LIN {X 0,Y 410.972,Z 398.401,A -85,B 0,C 180,E1 -10552.131,E2 -10552.131} C_VEL
LIN {X 0,Y 410.999,Z 397.235,A -85,B 0,C 180,E1 -10552.341,E2 -10552.341} C_VEL
LIN {X 0,Y 411.344,Z 382.792,A -85,B 0,C 180,E1 -10556.102,E2 -10556.102} C_VEL
LIN {X 0,Y 411.817,Z 369.639,A -85,B 0,C 180,E1 -10559.664,E2 -10559.664} C_VEL
LIN {X 0,Y 412.354,Z 356.779,A -85,B 0,C 180,E1 -10563.37,E2 -10563.37} C_VEL
LIN {X 0,Y 413.561,Z 344.278,A -85,B 0,C 180,E1 -10567.276,E2 -10567.276} C_VEL
LIN {X 0,Y 414.274,Z 339.521,A -85,B 0,C 180,E1 -10568.881,E2 -10568.881} C_VEL
LIN {X 0,Y 414.062,Z 336.041,A -85,B 0,C 180,E1 -10570.2,E2 -10570.2} C_VEL
LIN {X 0,Y 412.867,Z 329.754,A -85,B 0,C 180,E1 -10572.949,E2 -10572.949} C_VEL
LIN {X 0,Y 411.688,Z 324.313,A -85,B 0,C 180,E1 -10575.807,E2 -10575.807} C_VEL
LIN {X 0,Y 411.209,Z 321.929,A -85,B 0,C 180,E1 -10577.301,E2 -10577.301} C_VEL
LIN {X 0,Y 411.234,Z 321.886,A -85,B 0,C 180,E1 -10580.778,E2 -10580.778} C_VEL
LIN {X 0,Y 411.203,Z 321.888,A -85,B 0,C 180,E1 -10584.472,E2 -10584.472} C_VEL
LIN {X 0,Y 411.21,Z 321.889,A -85,B 0,C 180,E1 -10586.874,E2 -10586.874} C_VEL
LIN {X 0,Y 411.236,Z 321.885,A -85,B 0,C 180,E1 -10590.645,E2 -10590.645} C_VEL
LIN {X 0,Y 411.241,Z 321.886,A -85,B 0,C 180,E1 -10593.62,E2 -10593.62} C_VEL
LIN {X 0,Y 411.207,Z 321.891,A -85,B 0,C 180,E1 -10596.853,E2 -10596.853} C_VEL
LIN {X 0,Y 411.235,Z 322.056,A -85,B 0,C 180,E1 -10597.53,E2 -10597.53} C_VEL
LIN {X 0,Y 411.571,Z 323.361,A -85,B 0,C 180,E1 -10597.754,E2 -10597.754} C_VEL
LIN {X 0,Y 416.935,Z 335.703,A -85,B 0,C 180,E1 -10598.946,E2 -10598.946} C_VEL
LIN {X 0,Y 419.583,Z 343.599,A -85,B 0,C 180,E1 -10599.719,E2 -10599.719} C_VEL
LIN {X 0,Y 418.83,Z 355.331,A -85,B 0,C 180,E1 -10600.646,E2 -10600.646} C_VEL
LIN {X 0,Y 417.749,Z 367.989,A -85,B 0,C 180,E1 -10601.867,E2 -10601.867} C_VEL
LIN {X 0,Y 416.783,Z 378.362,A -85,B 0,C 180,E1 -10603.09,E2 -10603.09} C_VEL
LIN {X 0,Y 415.804,Z 388.025,A -85,B 0,C 180,E1 -10604.457,E2 -10604.457} C_VEL
LIN {X 0,Y 414.968,Z 394.51,A -85,B 0,C 180,E1 -10605.534,E2 -10605.534} C_VEL
LIN {X 0,Y 414.04,Z 403.147,A -85,B 0,C 180,E1 -10607.252,E2 -10607.252} C_VEL
LIN {X 0,Y 413.307,Z 409.172,A -85,B 0,C 180,E1 -10608.723,E2 -10608.723} C_VEL
LIN {X 0,Y 412.749,Z 414.131,A -85,B 0,C 180,E1 -10610.197,E2 -10610.197} C_VEL
LIN {X 0,Y 412.146,Z 419.249,A -85,B 0,C 180,E1 -10612.16,E2 -10612.16} C_VEL
LIN {X 0,Y 411.574,Z 422.875,A -85,B 0,C 180,E1 -10614.12,E2 -10614.12} C_VEL
LIN {X 0,Y 411.29,Z 425.054,A -85,B 0,C 180,E1 -10616.081,E2 -10616.081} C_VEL
LIN {X 0,Y 411.179,Z 425.847,A -85,B 0,C 180,E1 -10618.041,E2 -10618.041} C_VEL
LIN {X 0,Y 411.073,Z 425.319,A -85,B 0,C 180,E1 -10620,E2 -10620} C_VEL
LIN {X 0,Y 411.066,Z 423.45,A -85,B 0,C 180,E1 -10621.96,E2 -10621.96} C_VEL
LIN {X 0,Y 411.103,Z 420.216,A -85,B 0,C 180,E1 -10623.921,E2 -10623.921} C_VEL
LIN {X 0,Y 411.471,Z 415.498,A -85,B 0,C 180,E1 -10625.882,E2 -10625.882} C_VEL
LIN {X 0,Y 411.831,Z 410.884,A -85,B 0,C 180,E1 -10627.354,E2 -10627.354} C_VEL
LIN {X 0,Y 412.243,Z 404.257,A -85,B 0,C 180,E1 -10629.073,E2 -10629.073} C_VEL
LIN {X 0,Y 412.88,Z 396.057,A -85,B 0,C 180,E1 -10630.792,E2 -10630.792} C_VEL
LIN {X 0,Y 413.504,Z 387.517,A -85,B 0,C 180,E1 -10632.266,E2 -10632.266} C_VEL
LIN {X 0,Y 414.234,Z 377.269,A -85,B 0,C 180,E1 -10633.741,E2 -10633.741} C_VEL
LIN {X 0,Y 415.128,Z 365.737,A -85,B 0,C 180,E1 -10635.099,E2 -10635.099} C_VEL
LIN {X 0,Y 415.874,Z 353.184,A -85,B 0,C 180,E1 -10636.317,E2 -10636.317} C_VEL
LIN {X 0,Y 416.618,Z 341.348,A -85,B 0,C 180,E1 -10637.253,E2 -10637.253} C_VEL
LIN {X 0,Y 416.273,Z 338.757,A -85,B 0,C 180,E1 -10637.46,E2 -10637.46} C_VEL
LIN {X 0,Y 412.31,Z 325.603,A -85,B 0,C 180,E1 -10638.462,E2 -10638.462} C_VEL
LIN {X 0,Y 411.361,Z 322.465,A -85,B 0,C 180,E1 -10638.716,E2 -10638.716} C_VEL
LIN {X 0,Y 411.252,Z 321.899,A -85,B 0,C 180,E1 -10638.948,E2 -10638.948} C_VEL
LIN {X 0,Y 411.209,Z 321.891,A -85,B 0,C 180,E1 -10642.643,E2 -10642.643} C_VEL
LIN {X 0,Y 411.241,Z 321.881,A -85,B 0,C 180,E1 -10645.293,E2 -10645.293} C_VEL
LIN {X 0,Y 411.264,Z 321.877,A -85,B 0,C 180,E1 -10647.478,E2 -10647.478} C_VEL
LIN {X 0,Y 411.195,Z 321.89,A -85,B 0,C 180,E1 -10650.848,E2 -10650.848} C_VEL
LIN {X 0,Y 411.211,Z 321.888,A -85,B 0,C 180,E1 -10654.333,E2 -10654.333} C_VEL
LIN {X 0,Y 411.197,Z 321.887,A -85,B 0,C 180,E1 -10657.974,E2 -10657.974} C_VEL
LIN {X 0,Y 411.168,Z 321.889,A -85,B 0,C 180,E1 -10661.228,E2 -10661.228} C_VEL
LIN {X 0,Y 411.182,Z 321.894,A -85,B 0,C 180,E1 -10664.49,E2 -10664.49} C_VEL
LIN {X 0,Y 411.203,Z 321.89,A -85,B 0,C 180,E1 -10668.197,E2 -10668.197} C_VEL
LIN {X 0,Y 411.23,Z 321.884,A -85,B 0,C 180,E1 -10670.776,E2 -10670.776} C_VEL
LIN {X 0,Y 411.204,Z 321.889,A -85,B 0,C 180,E1 -10674.471,E2 -10674.471} C_VEL
LIN {X 0,Y 411.213,Z 321.884,A -85,B 0,C 180,E1 -10676.873,E2 -10676.873} C_VEL
LIN {X 0,Y 411.239,Z 321.882,A -85,B 0,C 180,E1 -10680.644,E2 -10680.644} C_VEL
LIN {X 0,Y 411.243,Z 321.881,A -85,B 0,C 180,E1 -10683.619,E2 -10683.619} C_VEL
LIN {X 0,Y 411.202,Z 321.885,A -85,B 0,C 180,E1 -10686.852,E2 -10686.852} C_VEL
LIN {X 0,Y 411.222,Z 321.89,A -85,B 0,C 180,E1 -10690.049,E2 -10690.049} C_VEL
LIN {X 0,Y 411.269,Z 321.877,A -85,B 0,C 180,E1 -10693.131,E2 -10693.131} C_VEL
LIN {X 0,Y 411.311,Z 321.871,A -85,B 0,C 180,E1 -10696.895,E2 -10696.895} C_VEL
LIN {X 0,Y 411.298,Z 321.877,A -85,B 0,C 180,E1 -10700.161,E2 -10700.161} C_VEL
LIN {X 0,Y 411.488,Z 321.853,A -85,B 0,C 180,E1 -10702.146,E2 -10702.146} C_VEL
LIN {X 0,Y 411.478,Z 321.854,A -85,B 0,C 180,E1 -10704.117,E2 -10704.117} C_VEL
LIN {X 0,Y 411.516,Z 321.85,A -85,B 0,C 180,E1 -10708.042,E2 -10708.042} C_VEL
LIN {X 0,Y 411.645,Z 321.834,A -85,B 0,C 180,E1 -10709.999,E2 -10709.999} C_VEL
LIN {X 0,Y 411.463,Z 321.853,A -85,B 0,C 180,E1 -10712.936,E2 -10712.936} C_VEL
LIN {X 0,Y 411.465,Z 321.852,A -85,B 0,C 180,E1 -10716.866,E2 -10716.866} C_VEL
LIN {X 0,Y 411.297,Z 321.877,A -85,B 0,C 180,E1 -10719.838,E2 -10719.838} C_VEL
LIN {X 0,Y 411.291,Z 321.874,A -85,B 0,C 180,E1 -10722.601,E2 -10722.601} C_VEL
LIN {X 0,Y 410.65,Z 321.959,A -85,B 0,C 180,E1 -10723.419,E2 -10723.419} C_VEL
LIN {X 0,Y 407.769,Z 322.313,A -85,B 0,C 180,E1 -10724.745,E2 -10724.745} C_VEL
LIN {X 0,Y 405.323,Z 322.621,A -85,B 0,C 180,E1 -10725.817,E2 -10725.817} C_VEL
LIN {X 0,Y 404.289,Z 322.747,A -85,B 0,C 180,E1 -10726.647,E2 -10726.647} C_VEL
LIN {X 0,Y 404.215,Z 322.757,A -85,B 0,C 180,E1 -10726.928,E2 -10726.928} C_VEL
LIN {X 0,Y 404.166,Z 322.761,A -85,B 0,C 180,E1 -10730.35,E2 -10730.35} C_VEL
LIN {X 0,Y 404.171,Z 322.766,A -85,B 0,C 180,E1 -10733.573,E2 -10733.573} C_VEL
LIN {X 0,Y 404.185,Z 322.762,A -85,B 0,C 180,E1 -10735.765,E2 -10735.765} C_VEL
LIN {X 0,Y 404.195,Z 322.758,A -85,B 0,C 180,E1 -10737.998,E2 -10737.998} C_VEL
LIN {X 0,Y 404.139,Z 322.768,A -85,B 0,C 180,E1 -10741.557,E2 -10741.557} C_VEL
LIN {X 0,Y 404.183,Z 322.764,A -85,B 0,C 180,E1 -10745.015,E2 -10745.015} C_VEL
LIN {X 0,Y 404.154,Z 322.766,A -85,B 0,C 180,E1 -10748.756,E2 -10748.756} C_VEL
LIN {X 0,Y 404.122,Z 322.769,A -85,B 0,C 180,E1 -10751.599,E2 -10751.599} C_VEL
LIN {X 0,Y 404.147,Z 322.765,A -85,B 0,C 180,E1 -10754.522,E2 -10754.522} C_VEL
LIN {X 0,Y 404.136,Z 322.769,A -85,B 0,C 180,E1 -10757.295,E2 -10757.295} C_VEL
LIN {X 0,Y 404.164,Z 322.761,A -85,B 0,C 180,E1 -10759.954,E2 -10759.954} C_VEL
LIN {X 0,Y 404.136,Z 322.77,A -85,B 0,C 180,E1 -10763.123,E2 -10763.123} C_VEL
LIN {X 0,Y 404.14,Z 322.765,A -85,B 0,C 180,E1 -10766.187,E2 -10766.187} C_VEL
LIN {X 0,Y 404.151,Z 322.763,A -85,B 0,C 180,E1 -10769.715,E2 -10769.715} C_VEL
LIN {X 0,Y 404.189,Z 322.762,A -85,B 0,C 180,E1 -10773.122,E2 -10773.122} C_VEL
LIN {X 0,Y 404.171,Z 322.762,A -85,B 0,C 180,E1 -10775.334,E2 -10775.334} C_VEL
LIN {X 0,Y 404.153,Z 322.769,A -85,B 0,C 180,E1 -10778.581,E2 -10778.581} C_VEL
LIN {X 0,Y 404.203,Z 322.757,A -85,B 0,C 180,E1 -10781.761,E2 -10781.761} C_VEL
LIN {X 0,Y 404.2,Z 322.761,A -85,B 0,C 180,E1 -10784.881,E2 -10784.881} C_VEL
LIN {X 0,Y 404.249,Z 322.752,A -85,B 0,C 180,E1 -10787.958,E2 -10787.958} C_VEL
LIN {X 0,Y 404.425,Z 322.732,A -85,B 0,C 180,E1 -10792.099,E2 -10792.099} C_VEL
LIN {X 0,Y 404.416,Z 322.732,A -85,B 0,C 180,E1 -10794.015,E2 -10794.015} C_VEL
LIN {X 0,Y 404.475,Z 322.725,A -85,B 0,C 180,E1 -10798.008,E2 -10798.008} C_VEL
LIN {X 0,Y 404.603,Z 322.71,A -85,B 0,C 180,E1 -10800,E2 -10800} C_VEL
LIN {X 0,Y 404.416,Z 322.731,A -85,B 0,C 180,E1 -10802.988,E2 -10802.988} C_VEL
LIN {X 0,Y 404.403,Z 322.732,A -85,B 0,C 180,E1 -10806.987,E2 -10806.987} C_VEL
LIN {X 0,Y 404.263,Z 322.754,A -85,B 0,C 180,E1 -10810.011,E2 -10810.011} C_VEL
LIN {X 0,Y 404.258,Z 322.75,A -85,B 0,C 180,E1 -10813.211,E2 -10813.211} C_VEL
LIN {X 0,Y 404.21,Z 322.756,A -85,B 0,C 180,E1 -10817.009,E2 -10817.009} C_VEL
LIN {X 0,Y 404.155,Z 322.766,A -85,B 0,C 180,E1 -10820.352,E2 -10820.352} C_VEL
LIN {X 0,Y 404.162,Z 322.764,A -85,B 0,C 180,E1 -10823.575,E2 -10823.575} C_VEL
LIN {X 0,Y 404.176,Z 322.765,A -85,B 0,C 180,E1 -10825.767,E2 -10825.767} C_VEL
LIN {X 0,Y 404.19,Z 322.765,A -85,B 0,C 180,E1 -10828,E2 -10828} C_VEL
LIN {X 0,Y 404.14,Z 322.768,A -85,B 0,C 180,E1 -10831.56,E2 -10831.56} C_VEL
LIN {X 0,Y 404.179,Z 322.76,A -85,B 0,C 180,E1 -10835.017,E2 -10835.017} C_VEL
LIN {X 0,Y 404.157,Z 322.767,A -85,B 0,C 180,E1 -10838.756,E2 -10838.756} C_VEL
LIN {X 0,Y 404.191,Z 322.962,A -85,B 0,C 180,E1 -10842.326,E2 -10842.326} C_VEL
LIN {X 0,Y 406.394,Z 333.763,A -85,B 0,C 180,E1 -10846.234,E2 -10846.234} C_VEL
LIN {X 0,Y 408.182,Z 342.533,A -85,B 0,C 180,E1 -10849.251,E2 -10849.251} C_VEL
LIN {X 0,Y 408.476,Z 347.13,A -85,B 0,C 180,E1 -10850.736,E2 -10850.736} C_VEL
LIN {X 0,Y 407.187,Z 360.221,A -85,B 0,C 180,E1 -10854.725,E2 -10854.725} C_VEL
LIN {X 0,Y 406.079,Z 373.732,A -85,B 0,C 180,E1 -10858.722,E2 -10858.722} C_VEL
LIN {X 0,Y 405.3,Z 385.351,A -85,B 0,C 180,E1 -10862.085,E2 -10862.085} C_VEL
LIN {X 0,Y 404.686,Z 396.904,A -85,B 0,C 180,E1 -10865.369,E2 -10865.369} C_VEL
LIN {X 0,Y 404.088,Z 408.948,A -85,B 0,C 180,E1 -10868.704,E2 -10868.704} C_VEL
LIN {X 0,Y 404.387,Z 411.516,A -85,B 0,C 180,E1 -10868.832,E2 -10868.832} C_VEL
LIN {X 0,Y 406.377,Z 426.794,A -85,B 0,C 180,E1 -10869.406,E2 -10869.406} C_VEL
LIN {X 0,Y 407.897,Z 440.761,A -85,B 0,C 180,E1 -10870.107,E2 -10870.107} C_VEL
LIN {X 0,Y 408.676,Z 451.116,A -85,B 0,C 180,E1 -10870.734,E2 -10870.734} C_VEL
LIN {X 0,Y 407.683,Z 464.047,A -85,B 0,C 180,E1 -10871.639,E2 -10871.639} C_VEL
LIN {X 0,Y 406.699,Z 477.124,A -85,B 0,C 180,E1 -10872.788,E2 -10872.788} C_VEL
LIN {X 0,Y 405.639,Z 488.756,A -85,B 0,C 180,E1 -10874.036,E2 -10874.036} C_VEL
LIN {X 0,Y 404.825,Z 499.405,A -85,B 0,C 180,E1 -10875.421,E2 -10875.421} C_VEL
LIN {X 0,Y 404.157,Z 509.073,A -85,B 0,C 180,E1 -10876.936,E2 -10876.936} C_VEL
LIN {X 0,Y 403.711,Z 518.347,A -85,B 0,C 180,E1 -10878.707,E2 -10878.707} C_VEL
LIN {X 0,Y 403.467,Z 525.787,A -85,B 0,C 180,E1 -10880.476,E2 -10880.476} C_VEL
LIN {X 0,Y 403.415,Z 530.976,A -85,B 0,C 180,E1 -10881.99,E2 -10881.99} C_VEL
LIN {X 0,Y 403.447,Z 534.312,A -85,B 0,C 180,E1 -10883.184,E2 -10883.184} C_VEL
LIN {X 0,Y 403.524,Z 538.294,A -85,B 0,C 180,E1 -10885.005,E2 -10885.005} C_VEL
LIN {X 0,Y 403.583,Z 539.923,A -85,B 0,C 180,E1 -10886.007,E2 -10886.007} C_VEL
LIN {X 0,Y 403.624,Z 542.027,A -85,B 0,C 180,E1 -10888.005,E2 -10888.005} C_VEL
LIN {X 0,Y 403.866,Z 542.674,A -85,B 0,C 180,E1 -10890.001,E2 -10890.001} C_VEL
LIN {X 0,Y 403.853,Z 542.423,A -85,B 0,C 180,E1 -10890.998,E2 -10890.998} C_VEL
LIN {X 0,Y 403.643,Z 540.784,A -85,B 0,C 180,E1 -10892.995,E2 -10892.995} C_VEL
LIN {X 0,Y 403.665,Z 539.422,A -85,B 0,C 180,E1 -10893.994,E2 -10893.994} C_VEL
LIN {X 0,Y 403.584,Z 536.612,A -85,B 0,C 180,E1 -10895.497,E2 -10895.497} C_VEL
LIN {X 0,Y 403.484,Z 532.933,A -85,B 0,C 180,E1 -10897.004,E2 -10897.004} C_VEL
LIN {X 0,Y 403.459,Z 528.291,A -85,B 0,C 180,E1 -10898.516,E2 -10898.516} C_VEL
LIN {X 0,Y 403.529,Z 521.585,A -85,B 0,C 180,E1 -10900.284,E2 -10900.284} C_VEL
LIN {X 0,Y 403.865,Z 513.357,A -85,B 0,C 180,E1 -10902.054,E2 -10902.054} C_VEL
LIN {X 0,Y 404.348,Z 505.162,A -85,B 0,C 180,E1 -10903.52,E2 -10903.52} C_VEL
LIN {X 0,Y 405.07,Z 494.839,A -85,B 0,C 180,E1 -10905.086,E2 -10905.086} C_VEL
LIN {X 0,Y 405.98,Z 483.957,A -85,B 0,C 180,E1 -10906.468,E2 -10906.468} C_VEL
LIN {X 0,Y 407.116,Z 470.983,A -85,B 0,C 180,E1 -10907.844,E2 -10907.844} C_VEL
LIN {X 0,Y 408.584,Z 456.723,A -85,B 0,C 180,E1 -10909.076,E2 -10909.076} C_VEL
LIN {X 0,Y 409.082,Z 450.098,A -85,B 0,C 180,E1 -10909.574,E2 -10909.574} C_VEL
LIN {X 0,Y 408.617,Z 436.574,A -85,B 0,C 180,E1 -10910.524,E2 -10910.524} C_VEL
LIN {X 0,Y 408.001,Z 422.468,A -85,B 0,C 180,E1 -10911.353,E2 -10911.353} C_VEL
LIN {X 0,Y 406.615,Z 410.859,A -85,B 0,C 180,E1 -10911.974,E2 -10911.974} C_VEL
LIN {X 0,Y 403.999,Z 396.607,A -85,B 0,C 180,E1 -10912.724,E2 -10912.724} C_VEL
LIN {X 0,Y 403.988,Z 394.774,A -85,B 0,C 180,E1 -10913.125,E2 -10913.125} C_VEL
LIN {X 0,Y 404.348,Z 381.832,A -85,B 0,C 180,E1 -10916.588,E2 -10916.588} C_VEL
LIN {X 0,Y 404.805,Z 370.429,A -85,B 0,C 180,E1 -10919.765,E2 -10919.765} C_VEL
LIN {X 0,Y 405.309,Z 359.068,A -85,B 0,C 180,E1 -10923.108,E2 -10923.108} C_VEL
LIN {X 0,Y 406.625,Z 345.801,A -85,B 0,C 180,E1 -10927.34,E2 -10927.34} C_VEL
LIN {X 0,Y 407.402,Z 340.779,A -85,B 0,C 180,E1 -10929.078,E2 -10929.078} C_VEL
LIN {X 0,Y 407.073,Z 337.024,A -85,B 0,C 180,E1 -10930.567,E2 -10930.567} C_VEL
LIN {X 0,Y 405.885,Z 330.926,A -85,B 0,C 180,E1 -10933.345,E2 -10933.345} C_VEL
LIN {X 0,Y 404.823,Z 326.031,A -85,B 0,C 180,E1 -10936.019,E2 -10936.019} C_VEL
LIN {X 0,Y 404.159,Z 322.794,A -85,B 0,C 180,E1 -10938.185,E2 -10938.185} C_VEL
LIN {X 0,Y 404.165,Z 322.768,A -85,B 0,C 180,E1 -10941.491,E2 -10941.491} C_VEL
LIN {X 0,Y 404.189,Z 322.763,A -85,B 0,C 180,E1 -10944.984,E2 -10944.984} C_VEL
LIN {X 0,Y 404.145,Z 322.767,A -85,B 0,C 180,E1 -10948.554,E2 -10948.554} C_VEL
LIN {X 0,Y 404.199,Z 322.763,A -85,B 0,C 180,E1 -10952.001,E2 -10952.001} C_VEL
LIN {X 0,Y 404.181,Z 322.765,A -85,B 0,C 180,E1 -10955.335,E2 -10955.335} C_VEL
LIN {X 0,Y 404.2,Z 322.912,A -85,B 0,C 180,E1 -10956.908,E2 -10956.908} C_VEL
LIN {X 0,Y 404.547,Z 324.306,A -85,B 0,C 180,E1 -10957.155,E2 -10957.155} C_VEL
LIN {X 0,Y 409.239,Z 334.539,A -85,B 0,C 180,E1 -10958.206,E2 -10958.206} C_VEL
LIN {X 0,Y 413.136,Z 345.425,A -85,B 0,C 180,E1 -10959.33,E2 -10959.33} C_VEL
LIN {X 0,Y 413.22,Z 347.8,A -85,B 0,C 180,E1 -10959.529,E2 -10959.529} C_VEL
LIN {X 0,Y 412.221,Z 360.274,A -85,B 0,C 180,E1 -10960.582,E2 -10960.582} C_VEL
LIN {X 0,Y 411.021,Z 372.151,A -85,B 0,C 180,E1 -10961.817,E2 -10961.817} C_VEL
LIN {X 0,Y 409.798,Z 383.765,A -85,B 0,C 180,E1 -10963.306,E2 -10963.306} C_VEL
LIN {X 0,Y 408.594,Z 393.394,A -85,B 0,C 180,E1 -10964.807,E2 -10964.807} C_VEL
LIN {X 0,Y 407.521,Z 402.396,A -85,B 0,C 180,E1 -10966.537,E2 -10966.537} C_VEL
LIN {X 0,Y 406.709,Z 408.757,A -85,B 0,C 180,E1 -10968.032,E2 -10968.032} C_VEL
LIN {X 0,Y 406.055,Z 413.979,A -85,B 0,C 180,E1 -10969.529,E2 -10969.529} C_VEL
LIN {X 0,Y 405.524,Z 418.29,A -85,B 0,C 180,E1 -10971.062,E2 -10971.062} C_VEL
LIN {X 0,Y 404.936,Z 422.493,A -85,B 0,C 180,E1 -10973.022,E2 -10973.022} C_VEL
LIN {X 0,Y 404.408,Z 425.339,A -85,B 0,C 180,E1 -10975.015,E2 -10975.015} C_VEL
LIN {X 0,Y 404.201,Z 426.748,A -85,B 0,C 180,E1 -10977.01,E2 -10977.01} C_VEL
LIN {X 0,Y 404.107,Z 426.82,A -85,B 0,C 180,E1 -10979.004,E2 -10979.004} C_VEL
LIN {X 0,Y 404.005,Z 425.57,A -85,B 0,C 180,E1 -10980.997,E2 -10980.997} C_VEL
LIN {X 0,Y 403.961,Z 422.971,A -85,B 0,C 180,E1 -10982.992,E2 -10982.992} C_VEL
LIN {X 0,Y 404.254,Z 418.934,A -85,B 0,C 180,E1 -10984.987,E2 -10984.987} C_VEL
LIN {X 0,Y 404.678,Z 413.372,A -85,B 0,C 180,E1 -10986.983,E2 -10986.983} C_VEL
LIN {X 0,Y 405.099,Z 407.779,A -85,B 0,C 180,E1 -10988.548,E2 -10988.548} C_VEL
LIN {X 0,Y 405.629,Z 400.47,A -85,B 0,C 180,E1 -10990.23,E2 -10990.23} C_VEL
LIN {X 0,Y 406.3,Z 391.111,A -85,B 0,C 180,E1 -10991.98,E2 -10991.98} C_VEL
LIN {X 0,Y 407.009,Z 381.355,A -85,B 0,C 180,E1 -10993.481,E2 -10993.481} C_VEL
LIN {X 0,Y 407.903,Z 370.599,A -85,B 0,C 180,E1 -10994.85,E2 -10994.85} C_VEL
LIN {X 0,Y 408.742,Z 358.809,A -85,B 0,C 180,E1 -10996.097,E2 -10996.097} C_VEL
LIN {X 0,Y 409.514,Z 347.643,A -85,B 0,C 180,E1 -10997.072,E2 -10997.072} C_VEL
LIN {X 0,Y 409.769,Z 342.118,A -85,B 0,C 180,E1 -10997.495,E2 -10997.495} C_VEL
LIN {X 0,Y 406.145,Z 329.28,A -85,B 0,C 180,E1 -10998.525,E2 -10998.525} C_VEL
LIN {X 0,Y 404.313,Z 323.32,A -85,B 0,C 180,E1 -10998.989,E2 -10998.989} C_VEL
LIN {X 0,Y 404.205,Z 322.802,A -85,B 0,C 180,E1 -10999.159,E2 -10999.159} C_VEL
LIN {X 0,Y 404.161,Z 322.769,A -85,B 0,C 180,E1 -11002.834,E2 -11002.834} C_VEL
LIN {X 0,Y 404.189,Z 322.758,A -85,B 0,C 180,E1 -11005.766,E2 -11005.766} C_VEL
LIN {X 0,Y 404.2,Z 322.758,A -85,B 0,C 180,E1 -11008,E2 -11008} C_VEL
LIN {X 0,Y 404.144,Z 322.764,A -85,B 0,C 180,E1 -11011.558,E2 -11011.558} C_VEL
LIN {X 0,Y 404.19,Z 322.761,A -85,B 0,C 180,E1 -11015.016,E2 -11015.016} C_VEL
LIN {X 0,Y 404.156,Z 322.767,A -85,B 0,C 180,E1 -11018.757,E2 -11018.757} C_VEL
LIN {X 0,Y 404.128,Z 322.766,A -85,B 0,C 180,E1 -11021.6,E2 -11021.6} C_VEL
LIN {X 0,Y 404.152,Z 322.769,A -85,B 0,C 180,E1 -11024.522,E2 -11024.522} C_VEL
LIN {X 0,Y 404.179,Z 322.76,A -85,B 0,C 180,E1 -11027.3,E2 -11027.3} C_VEL
LIN {X 0,Y 404.175,Z 322.763,A -85,B 0,C 180,E1 -11029.955,E2 -11029.955} C_VEL
LIN {X 0,Y 404.144,Z 322.764,A -85,B 0,C 180,E1 -11033.124,E2 -11033.124} C_VEL
LIN {X 0,Y 404.151,Z 322.77,A -85,B 0,C 180,E1 -11036.187,E2 -11036.187} C_VEL
LIN {X 0,Y 404.152,Z 322.765,A -85,B 0,C 180,E1 -11039.715,E2 -11039.715} C_VEL
LIN {X 0,Y 404.201,Z 322.757,A -85,B 0,C 180,E1 -11043.122,E2 -11043.122} C_VEL
LIN {X 0,Y 404.18,Z 322.76,A -85,B 0,C 180,E1 -11045.334,E2 -11045.334} C_VEL
LIN {X 0,Y 404.145,Z 322.766,A -85,B 0,C 180,E1 -11048.58,E2 -11048.58} C_VEL
LIN {X 0,Y 404.217,Z 322.759,A -85,B 0,C 180,E1 -11051.761,E2 -11051.761} C_VEL
LIN {X 0,Y 404.212,Z 322.756,A -85,B 0,C 180,E1 -11054.881,E2 -11054.881} C_VEL
LIN {X 0,Y 404.262,Z 322.756,A -85,B 0,C 180,E1 -11057.958,E2 -11057.958} C_VEL
LIN {X 0,Y 404.439,Z 322.732,A -85,B 0,C 180,E1 -11062.099,E2 -11062.099} C_VEL
LIN {X 0,Y 404.427,Z 322.734,A -85,B 0,C 180,E1 -11064.014,E2 -11064.014} C_VEL
LIN {X 0,Y 404.485,Z 322.726,A -85,B 0,C 180,E1 -11068.008,E2 -11068.008} C_VEL
LIN {X 0,Y 404.615,Z 322.71,A -85,B 0,C 180,E1 -11069.999,E2 -11069.999} C_VEL
LIN {X 0,Y 404.421,Z 322.73,A -85,B 0,C 180,E1 -11072.987,E2 -11072.987} C_VEL
LIN {X 0,Y 404.416,Z 322.731,A -85,B 0,C 180,E1 -11076.986,E2 -11076.986} C_VEL
LIN {X 0,Y 404.262,Z 322.752,A -85,B 0,C 180,E1 -11080.011,E2 -11080.011} C_VEL
LIN {X 0,Y 404.269,Z 322.752,A -85,B 0,C 180,E1 -11083.21,E2 -11083.21} C_VEL
LIN {X 0,Y 404.215,Z 322.757,A -85,B 0,C 180,E1 -11086.928,E2 -11086.928} C_VEL
LIN {X 0,Y 403.564,Z 322.843,A -85,B 0,C 180,E1 -11087.76,E2 -11087.76} C_VEL
LIN {X 0,Y 400.677,Z 323.2,A -85,B 0,C 180,E1 -11089.111,E2 -11089.111} C_VEL
LIN {X 0,Y 398.222,Z 323.502,A -85,B 0,C 180,E1 -11090.203,E2 -11090.203} C_VEL
LIN {X 0,Y 397.174,Z 323.635,A -85,B 0,C 180,E1 -11091.048,E2 -11091.048} C_VEL
LIN {X 0,Y 397.093,Z 323.642,A -85,B 0,C 180,E1 -11091.334,E2 -11091.334} C_VEL
LIN {X 0,Y 397.134,Z 323.638,A -85,B 0,C 180,E1 -11094.017,E2 -11094.017} C_VEL
LIN {X 0,Y 397.195,Z 323.636,A -85,B 0,C 180,E1 -11097.389,E2 -11097.389} C_VEL
LIN {X 0,Y 397.078,Z 323.647,A -85,B 0,C 180,E1 -11100.881,E2 -11100.881} C_VEL
LIN {X 0,Y 397.124,Z 323.639,A -85,B 0,C 180,E1 -11104.492,E2 -11104.492} C_VEL
LIN {X 0,Y 397.101,Z 323.641,A -85,B 0,C 180,E1 -11108.274,E2 -11108.274} C_VEL
LIN {X 0,Y 397.087,Z 323.648,A -85,B 0,C 180,E1 -11110.907,E2 -11110.907} C_VEL
LIN {X 0,Y 397.101,Z 323.643,A -85,B 0,C 180,E1 -11113.647,E2 -11113.647} C_VEL
LIN {X 0,Y 397.101,Z 323.643,A -85,B 0,C 180,E1 -11116.519,E2 -11116.519} C_VEL
LIN {X 0,Y 397.111,Z 323.642,A -85,B 0,C 180,E1 -11120.422,E2 -11120.422} C_VEL
LIN {X 0,Y 397.104,Z 323.642,A -85,B 0,C 180,E1 -11124.264,E2 -11124.264} C_VEL
LIN {X 0,Y 397.11,Z 323.645,A -85,B 0,C 180,E1 -11126.726,E2 -11126.726} C_VEL
LIN {X 0,Y 397.129,Z 323.639,A -85,B 0,C 180,E1 -11130.296,E2 -11130.296} C_VEL
LIN {X 0,Y 397.189,Z 323.635,A -85,B 0,C 180,E1 -11132.609,E2 -11132.609} C_VEL
LIN {X 0,Y 397.126,Z 323.639,A -85,B 0,C 180,E1 -11135.981,E2 -11135.981} C_VEL
LIN {X 0,Y 397.132,Z 323.638,A -85,B 0,C 180,E1 -11139.704,E2 -11139.704} C_VEL
LIN {X 0,Y 397.175,Z 323.637,A -85,B 0,C 180,E1 -11142.844,E2 -11142.844} C_VEL
LIN {X 0,Y 397.219,Z 323.633,A -85,B 0,C 180,E1 -11146.678,E2 -11146.678} C_VEL
LIN {X 0,Y 397.211,Z 323.628,A -85,B 0,C 180,E1 -11149.808,E2 -11149.808} C_VEL
LIN {X 0,Y 397.356,Z 323.612,A -85,B 0,C 180,E1 -11152.888,E2 -11152.888} C_VEL
LIN {X 0,Y 397.249,Z 323.625,A -85,B 0,C 180,E1 -11154.925,E2 -11154.925} C_VEL
LIN {X 0,Y 397.444,Z 323.601,A -85,B 0,C 180,E1 -11157.973,E2 -11157.973} C_VEL
LIN {X 0,Y 397.573,Z 323.585,A -85,B 0,C 180,E1 -11160,E2 -11160} C_VEL
LIN {X 0,Y 397.375,Z 323.608,A -85,B 0,C 180,E1 -11163.041,E2 -11163.041} C_VEL
LIN {X 0,Y 397.356,Z 323.61,A -85,B 0,C 180,E1 -11167.112,E2 -11167.112} C_VEL
LIN {X 0,Y 397.22,Z 323.633,A -85,B 0,C 180,E1 -11170.191,E2 -11170.191} C_VEL
LIN {X 0,Y 397.218,Z 323.627,A -85,B 0,C 180,E1 -11173.321,E2 -11173.321} C_VEL
LIN {X 0,Y 397.163,Z 323.637,A -85,B 0,C 180,E1 -11176.447,E2 -11176.447} C_VEL
LIN {X 0,Y 397.14,Z 323.639,A -85,B 0,C 180,E1 -11179.647,E2 -11179.647} C_VEL
LIN {X 0,Y 397.127,Z 323.638,A -85,B 0,C 180,E1 -11183.041,E2 -11183.041} C_VEL
LIN {X 0,Y 397.127,Z 323.642,A -85,B 0,C 180,E1 -11186.259,E2 -11186.259} C_VEL
LIN {X 0,Y 397.119,Z 323.64,A -85,B 0,C 180,E1 -11188.544,E2 -11188.544} C_VEL
LIN {X 0,Y 397.104,Z 323.646,A -85,B 0,C 180,E1 -11192.069,E2 -11192.069} C_VEL
LIN {X 0,Y 397.113,Z 323.643,A -85,B 0,C 180,E1 -11195.504,E2 -11195.504} C_VEL
LIN {X 0,Y 397.131,Z 323.642,A -85,B 0,C 180,E1 -11198.864,E2 -11198.864} C_VEL
LIN {X 0,Y 397.142,Z 323.797,A -85,B 0,C 180,E1 -11201.95,E2 -11201.95} C_VEL
LIN {X 0,Y 399.138,Z 333.65,A -85,B 0,C 180,E1 -11205.607,E2 -11205.607} C_VEL
LIN {X 0,Y 401.07,Z 342.994,A -85,B 0,C 180,E1 -11208.894,E2 -11208.894} C_VEL
LIN {X 0,Y 401.58,Z 347.385,A -85,B 0,C 180,E1 -11210.357,E2 -11210.357} C_VEL
LIN {X 0,Y 400.563,Z 357.066,A -85,B 0,C 180,E1 -11213.379,E2 -11213.379} C_VEL
LIN {X 0,Y 399.484,Z 368.797,A -85,B 0,C 180,E1 -11216.951,E2 -11216.951} C_VEL
LIN {X 0,Y 398.711,Z 379.218,A -85,B 0,C 180,E1 -11220.062,E2 -11220.062} C_VEL
LIN {X 0,Y 397.893,Z 391.981,A -85,B 0,C 180,E1 -11223.797,E2 -11223.797} C_VEL
LIN {X 0,Y 397.31,Z 403.457,A -85,B 0,C 180,E1 -11227.099,E2 -11227.099} C_VEL
LIN {X 0,Y 397.081,Z 408.159,A -85,B 0,C 180,E1 -11228.387,E2 -11228.387} C_VEL
LIN {X 0,Y 397.449,Z 411.657,A -85,B 0,C 180,E1 -11228.554,E2 -11228.554} C_VEL
LIN {X 0,Y 399.488,Z 427.529,A -85,B 0,C 180,E1 -11229.183,E2 -11229.183} C_VEL
LIN {X 0,Y 401.026,Z 442.061,A -85,B 0,C 180,E1 -11229.952,E2 -11229.952} C_VEL
LIN {X 0,Y 401.66,Z 451.942,A -85,B 0,C 180,E1 -11230.584,E2 -11230.584} C_VEL
LIN {X 0,Y 400.59,Z 465.561,A -85,B 0,C 180,E1 -11231.592,E2 -11231.592} C_VEL
LIN {X 0,Y 399.618,Z 477.962,A -85,B 0,C 180,E1 -11232.737,E2 -11232.737} C_VEL
LIN {X 0,Y 398.55,Z 489.292,A -85,B 0,C 180,E1 -11234.008,E2 -11234.008} C_VEL
LIN {X 0,Y 397.709,Z 499.693,A -85,B 0,C 180,E1 -11235.416,E2 -11235.416} C_VEL
LIN {X 0,Y 397.048,Z 509.046,A -85,B 0,C 180,E1 -11236.94,E2 -11236.94} C_VEL
LIN {X 0,Y 396.673,Z 517.028,A -85,B 0,C 180,E1 -11238.504,E2 -11238.504} C_VEL
LIN {X 0,Y 396.428,Z 524.544,A -85,B 0,C 180,E1 -11240.305,E2 -11240.305} C_VEL
LIN {X 0,Y 396.354,Z 529.758,A -85,B 0,C 180,E1 -11241.846,E2 -11241.846} C_VEL
LIN {X 0,Y 396.392,Z 533.371,A -85,B 0,C 180,E1 -11243.157,E2 -11243.157} C_VEL
LIN {X 0,Y 396.489,Z 537.166,A -85,B 0,C 180,E1 -11244.916,E2 -11244.916} C_VEL
LIN {X 0,Y 396.547,Z 538.811,A -85,B 0,C 180,E1 -11245.936,E2 -11245.936} C_VEL
LIN {X 0,Y 396.597,Z 540.944,A -85,B 0,C 180,E1 -11247.97,E2 -11247.97} C_VEL
LIN {X 0,Y 396.868,Z 541.619,A -85,B 0,C 180,E1 -11250.001,E2 -11250.001} C_VEL
LIN {X 0,Y 396.828,Z 541.372,A -85,B 0,C 180,E1 -11251.016,E2 -11251.016} C_VEL
LIN {X 0,Y 396.605,Z 539.743,A -85,B 0,C 180,E1 -11253.048,E2 -11253.048} C_VEL
LIN {X 0,Y 396.628,Z 538.39,A -85,B 0,C 180,E1 -11254.065,E2 -11254.065} C_VEL
LIN {X 0,Y 396.522,Z 535.594,A -85,B 0,C 180,E1 -11255.595,E2 -11255.595} C_VEL
LIN {X 0,Y 396.415,Z 530.477,A -85,B 0,C 180,E1 -11257.642,E2 -11257.642} C_VEL
LIN {X 0,Y 396.41,Z 523.666,A -85,B 0,C 180,E1 -11259.697,E2 -11259.697} C_VEL
LIN {X 0,Y 396.662,Z 516.148,A -85,B 0,C 180,E1 -11261.498,E2 -11261.498} C_VEL
LIN {X 0,Y 397.154,Z 506.961,A -85,B 0,C 180,E1 -11263.301,E2 -11263.301} C_VEL
LIN {X 0,Y 397.828,Z 497.544,A -85,B 0,C 180,E1 -11264.843,E2 -11264.843} C_VEL
LIN {X 0,Y 398.82,Z 486.388,A -85,B 0,C 180,E1 -11266.378,E2 -11266.378} C_VEL
LIN {X 0,Y 400.046,Z 473.024,A -85,B 0,C 180,E1 -11267.906,E2 -11267.906} C_VEL
LIN {X 0,Y 401.617,Z 459.068,A -85,B 0,C 180,E1 -11269.203,E2 -11269.203} C_VEL
LIN {X 0,Y 402.287,Z 450.086,A -85,B 0,C 180,E1 -11269.918,E2 -11269.918} C_VEL
LIN {X 0,Y 401.981,Z 436.828,A -85,B 0,C 180,E1 -11270.893,E2 -11270.893} C_VEL
LIN {X 0,Y 401.432,Z 422.551,A -85,B 0,C 180,E1 -11271.781,E2 -11271.781} C_VEL
LIN {X 0,Y 399.852,Z 409.684,A -85,B 0,C 180,E1 -11272.519,E2 -11272.519} C_VEL
LIN {X 0,Y 396.979,Z 394.949,A -85,B 0,C 180,E1 -11273.351,E2 -11273.351} C_VEL
LIN {X 0,Y 396.948,Z 394.098,A -85,B 0,C 180,E1 -11273.477,E2 -11273.477} C_VEL
LIN {X 0,Y 397.309,Z 381.941,A -85,B 0,C 180,E1 -11276.813,E2 -11276.813} C_VEL
LIN {X 0,Y 397.855,Z 369.52,A -85,B 0,C 180,E1 -11280.373,E2 -11280.373} C_VEL
LIN {X 0,Y 398.511,Z 357.601,A -85,B 0,C 180,E1 -11284.017,E2 -11284.017} C_VEL
LIN {X 0,Y 399.948,Z 345.752,A -85,B 0,C 180,E1 -11287.955,E2 -11287.955} C_VEL
LIN {X 0,Y 400.52,Z 341.61,A -85,B 0,C 180,E1 -11289.459,E2 -11289.459} C_VEL
LIN {X 0,Y 399.917,Z 337.103,A -85,B 0,C 180,E1 -11291.359,E2 -11291.359} C_VEL
LIN {X 0,Y 398.667,Z 330.924,A -85,B 0,C 180,E1 -11294.394,E2 -11294.394} C_VEL
LIN {X 0,Y 397.689,Z 326.355,A -85,B 0,C 180,E1 -11297.127,E2 -11297.127} C_VEL
LIN {X 0,Y 397.116,Z 323.672,A -85,B 0,C 180,E1 -11299.095,E2 -11299.095} C_VEL
LIN {X 0,Y 397.113,Z 323.645,A -85,B 0,C 180,E1 -11301.726,E2 -11301.726} C_VEL
LIN {X 0,Y 397.129,Z 323.643,A -85,B 0,C 180,E1 -11305.507,E2 -11305.507} C_VEL
LIN {X 0,Y 397.082,Z 323.648,A -85,B 0,C 180,E1 -11309.118,E2 -11309.118} C_VEL
LIN {X 0,Y 397.198,Z 323.635,A -85,B 0,C 180,E1 -11312.61,E2 -11312.61} C_VEL
LIN {X 0,Y 397.137,Z 323.73,A -85,B 0,C 180,E1 -11316.216,E2 -11316.216} C_VEL
LIN {X 0,Y 397.398,Z 324.834,A -85,B 0,C 180,E1 -11316.463,E2 -11316.463} C_VEL
LIN {X 0,Y 402.625,Z 336.052,A -85,B 0,C 180,E1 -11317.691,E2 -11317.691} C_VEL
LIN {X 0,Y 406.737,Z 347.286,A -85,B 0,C 180,E1 -11318.919,E2 -11318.919} C_VEL
LIN {X 0,Y 406.978,Z 349.373,A -85,B 0,C 180,E1 -11319.115,E2 -11319.115} C_VEL
LIN {X 0,Y 405.92,Z 361.226,A -85,B 0,C 180,E1 -11320.137,E2 -11320.137} C_VEL
LIN {X 0,Y 404.772,Z 372.04,A -85,B 0,C 180,E1 -11321.264,E2 -11321.264} C_VEL
LIN {X 0,Y 403.664,Z 382.067,A -85,B 0,C 180,E1 -11322.523,E2 -11322.523} C_VEL
LIN {X 0,Y 402.401,Z 392.127,A -85,B 0,C 180,E1 -11324.048,E2 -11324.048} C_VEL
LIN {X 0,Y 401.473,Z 399.078,A -85,B 0,C 180,E1 -11325.296,E2 -11325.296} C_VEL
LIN {X 0,Y 400.379,Z 407.222,A -85,B 0,C 180,E1 -11327.068,E2 -11327.068} C_VEL
LIN {X 0,Y 399.43,Z 413.77,A -85,B 0,C 180,E1 -11328.84,E2 -11328.84} C_VEL
LIN {X 0,Y 398.665,Z 419.54,A -85,B 0,C 180,E1 -11330.871,E2 -11330.871} C_VEL
LIN {X 0,Y 398,Z 423.772,A -85,B 0,C 180,E1 -11332.9,E2 -11332.9} C_VEL
LIN {X 0,Y 397.434,Z 426.544,A -85,B 0,C 180,E1 -11334.928,E2 -11334.928} C_VEL
LIN {X 0,Y 397.225,Z 427.883,A -85,B 0,C 180,E1 -11336.958,E2 -11336.958} C_VEL
LIN {X 0,Y 397.097,Z 427.893,A -85,B 0,C 180,E1 -11338.986,E2 -11338.986} C_VEL
LIN {X 0,Y 397.003,Z 426.576,A -85,B 0,C 180,E1 -11341.015,E2 -11341.015} C_VEL
LIN {X 0,Y 396.934,Z 423.915,A -85,B 0,C 180,E1 -11343.045,E2 -11343.045} C_VEL
LIN {X 0,Y 397.245,Z 419.807,A -85,B 0,C 180,E1 -11345.075,E2 -11345.075} C_VEL
LIN {X 0,Y 397.681,Z 414.357,A -85,B 0,C 180,E1 -11347.038,E2 -11347.038} C_VEL
LIN {X 0,Y 398.111,Z 408.648,A -85,B 0,C 180,E1 -11348.661,E2 -11348.661} C_VEL
LIN {X 0,Y 398.684,Z 401.109,A -85,B 0,C 180,E1 -11350.41,E2 -11350.41} C_VEL
LIN {X 0,Y 399.251,Z 393.142,A -85,B 0,C 180,E1 -11351.937,E2 -11351.937} C_VEL
LIN {X 0,Y 399.993,Z 383.588,A -85,B 0,C 180,E1 -11353.463,E2 -11353.463} C_VEL
LIN {X 0,Y 400.983,Z 371.996,A -85,B 0,C 180,E1 -11354.983,E2 -11354.983} C_VEL
LIN {X 0,Y 401.831,Z 360.297,A -85,B 0,C 180,E1 -11356.251,E2 -11356.251} C_VEL
LIN {X 0,Y 402.613,Z 349.017,A -85,B 0,C 180,E1 -11357.263,E2 -11357.263} C_VEL
LIN {X 0,Y 402.811,Z 342.824,A -85,B 0,C 180,E1 -11357.752,E2 -11357.752} C_VEL
LIN {X 0,Y 399.079,Z 330.189,A -85,B 0,C 180,E1 -11358.788,E2 -11358.788} C_VEL
LIN {X 0,Y 397.278,Z 324.391,A -85,B 0,C 180,E1 -11359.237,E2 -11359.237} C_VEL
LIN {X 0,Y 397.168,Z 323.676,A -85,B 0,C 180,E1 -11359.445,E2 -11359.445} C_VEL
LIN {X 0,Y 397.14,Z 323.643,A -85,B 0,C 180,E1 -11363.041,E2 -11363.041} C_VEL
LIN {X 0,Y 397.14,Z 323.639,A -85,B 0,C 180,E1 -11366.258,E2 -11366.258} C_VEL
LIN {X 0,Y 397.128,Z 323.644,A -85,B 0,C 180,E1 -11368.544,E2 -11368.544} C_VEL
LIN {X 0,Y 397.083,Z 323.645,A -85,B 0,C 180,E1 -11372.072,E2 -11372.072} C_VEL
LIN {X 0,Y 397.125,Z 323.638,A -85,B 0,C 180,E1 -11375.503,E2 -11375.503} C_VEL
LIN {X 0,Y 397.132,Z 323.641,A -85,B 0,C 180,E1 -11378.861,E2 -11378.861} C_VEL
LIN {X 0,Y 397.074,Z 323.65,A -85,B 0,C 180,E1 -11382.267,E2 -11382.267} C_VEL
LIN {X 0,Y 397.095,Z 323.643,A -85,B 0,C 180,E1 -11385.068,E2 -11385.068} C_VEL
LIN {X 0,Y 397.115,Z 323.643,A -85,B 0,C 180,E1 -11388.014,E2 -11388.014} C_VEL
LIN {X 0,Y 397.139,Z 323.637,A -85,B 0,C 180,E1 -11391.138,E2 -11391.138} C_VEL
LIN {X 0,Y 397.125,Z 323.643,A -85,B 0,C 180,E1 -11394.496,E2 -11394.496} C_VEL
LIN {X 0,Y 397.085,Z 323.647,A -85,B 0,C 180,E1 -11397.928,E2 -11397.928} C_VEL
LIN {X 0,Y 397.128,Z 323.639,A -85,B 0,C 180,E1 -11401.456,E2 -11401.456} C_VEL
LIN {X 0,Y 397.158,Z 323.637,A -85,B 0,C 180,E1 -11404.487,E2 -11404.487} C_VEL
LIN {X 0,Y 397.102,Z 323.647,A -85,B 0,C 180,E1 -11408.181,E2 -11408.181} C_VEL
LIN {X 0,Y 397.169,Z 323.634,A -85,B 0,C 180,E1 -11411.426,E2 -11411.426} C_VEL
LIN {X 0,Y 397.185,Z 323.632,A -85,B 0,C 180,E1 -11414.607,E2 -11414.607} C_VEL
LIN {X 0,Y 397.225,Z 323.631,A -85,B 0,C 180,E1 -11417.741,E2 -11417.741} C_VEL
LIN {X 0,Y 397.4,Z 323.609,A -85,B 0,C 180,E1 -11422.04,E2 -11422.04} C_VEL
LIN {X 0,Y 397.258,Z 323.622,A -85,B 0,C 180,E1 -11424.924,E2 -11424.924} C_VEL
LIN {X 0,Y 397.454,Z 323.602,A -85,B 0,C 180,E1 -11427.972,E2 -11427.972} C_VEL
LIN {X 0,Y 397.584,Z 323.585,A -85,B 0,C 180,E1 -11429.999,E2 -11429.999} C_VEL
LIN {X 0,Y 397.38,Z 323.607,A -85,B 0,C 180,E1 -11433.04,E2 -11433.04} C_VEL
LIN {X 0,Y 397.368,Z 323.61,A -85,B 0,C 180,E1 -11437.111,E2 -11437.111} C_VEL
LIN {X 0,Y 397.222,Z 323.628,A -85,B 0,C 180,E1 -11440.19,E2 -11440.19} C_VEL
LIN {X 0,Y 397.229,Z 323.63,A -85,B 0,C 180,E1 -11443.32,E2 -11443.32} C_VEL
LIN {X 0,Y 397.184,Z 323.634,A -85,B 0,C 180,E1 -11447.154,E2 -11447.154} C_VEL
LIN {X 0,Y 397.111,Z 323.641,A -85,B 0,C 180,E1 -11450.728,E2 -11450.728} C_VEL
LIN {X 0,Y 397.093,Z 323.642,A -85,B 0,C 180,E1 -11451.334,E2 -11451.334} C_VEL
LIN {X 0,Y 396.45,Z 323.725,A -85,B 0,C 180,E1 -11452.18,E2 -11452.18} C_VEL
LIN {X 0,Y 393.649,Z 324.079,A -85,B 0,C 180,E1 -11453.557,E2 -11453.557} C_VEL
LIN {X 0,Y 391.257,Z 324.377,A -85,B 0,C 180,E1 -11454.669,E2 -11454.669} C_VEL
LIN {X 0,Y 390.211,Z 324.505,A -85,B 0,C 180,E1 -11455.528,E2 -11455.528} C_VEL
LIN {X 0,Y 390.115,Z 324.514,A -85,B 0,C 180,E1 -11455.819,E2 -11455.819} C_VEL
LIN {X 0,Y 390.059,Z 324.523,A -85,B 0,C 180,E1 -11459.108,E2 -11459.108} C_VEL
LIN {X 0,Y 390.042,Z 324.522,A -85,B 0,C 180,E1 -11462.72,E2 -11462.72} C_VEL
LIN {X 0,Y 390.054,Z 324.52,A -85,B 0,C 180,E1 -11465.824,E2 -11465.824} C_VEL
LIN {X 0,Y 390.068,Z 324.524,A -85,B 0,C 180,E1 -11469.217,E2 -11469.217} C_VEL
LIN {X 0,Y 390.042,Z 324.521,A -85,B 0,C 180,E1 -11472.373,E2 -11472.373} C_VEL
LIN {X 0,Y 390.045,Z 324.524,A -85,B 0,C 180,E1 -11475.354,E2 -11475.354} C_VEL
LIN {X 0,Y 390.029,Z 324.523,A -85,B 0,C 180,E1 -11478.186,E2 -11478.186} C_VEL
LIN {X 0,Y 390.088,Z 324.521,A -85,B 0,C 180,E1 -11480.907,E2 -11480.907} C_VEL
LIN {X 0,Y 390.081,Z 324.521,A -85,B 0,C 180,E1 -11484.792,E2 -11484.792} C_VEL
LIN {X 0,Y 390.044,Z 324.523,A -85,B 0,C 180,E1 -11488.497,E2 -11488.497} C_VEL
LIN {X 0,Y 390.111,Z 324.513,A -85,B 0,C 180,E1 -11492.069,E2 -11492.069} C_VEL
LIN {X 0,Y 390.073,Z 324.517,A -85,B 0,C 180,E1 -11495.518,E2 -11495.518} C_VEL
LIN {X 0,Y 390.056,Z 324.524,A -85,B 0,C 180,E1 -11498.877,E2 -11498.877} C_VEL
LIN {X 0,Y 390.121,Z 324.513,A -85,B 0,C 180,E1 -11502.166,E2 -11502.166} C_VEL
LIN {X 0,Y 390.137,Z 324.509,A -85,B 0,C 180,E1 -11505.392,E2 -11505.392} C_VEL
LIN {X 0,Y 390.142,Z 324.515,A -85,B 0,C 180,E1 -11508.571,E2 -11508.571} C_VEL
LIN {X 0,Y 390.336,Z 324.486,A -85,B 0,C 180,E1 -11511.993,E2 -11511.993} C_VEL
LIN {X 0,Y 390.221,Z 324.501,A -85,B 0,C 180,E1 -11514.833,E2 -11514.833} C_VEL
LIN {X 0,Y 390.413,Z 324.477,A -85,B 0,C 180,E1 -11517.936,E2 -11517.936} C_VEL
LIN {X 0,Y 390.542,Z 324.461,A -85,B 0,C 180,E1 -11520,E2 -11520} C_VEL
LIN {X 0,Y 390.309,Z 324.488,A -85,B 0,C 180,E1 -11523.096,E2 -11523.096} C_VEL
LIN {X 0,Y 390.322,Z 324.492,A -85,B 0,C 180,E1 -11526.202,E2 -11526.202} C_VEL
LIN {X 0,Y 390.307,Z 324.495,A -85,B 0,C 180,E1 -11528.282,E2 -11528.282} C_VEL
LIN {X 0,Y 390.17,Z 324.509,A -85,B 0,C 180,E1 -11532.483,E2 -11532.483} C_VEL
LIN {X 0,Y 390.136,Z 324.511,A -85,B 0,C 180,E1 -11535.677,E2 -11535.677} C_VEL
LIN {X 0,Y 390.097,Z 324.514,A -85,B 0,C 180,E1 -11538.922,E2 -11538.922} C_VEL
LIN {X 0,Y 390.032,Z 324.527,A -85,B 0,C 180,E1 -11542.234,E2 -11542.234} C_VEL
LIN {X 0,Y 390.111,Z 324.516,A -85,B 0,C 180,E1 -11545.744,E2 -11545.744} C_VEL
LIN {X 0,Y 390.058,Z 324.519,A -85,B 0,C 180,E1 -11549.109,E2 -11549.109} C_VEL
LIN {X 0,Y 390.048,Z 324.52,A -85,B 0,C 180,E1 -11552.721,E2 -11552.721} C_VEL
LIN {X 0,Y 390.051,Z 324.527,A -85,B 0,C 180,E1 -11555.826,E2 -11555.826} C_VEL
LIN {X 0,Y 390.068,Z 324.523,A -85,B 0,C 180,E1 -11559.22,E2 -11559.22} C_VEL
LIN {X 0,Y 390.102,Z 324.668,A -85,B 0,C 180,E1 -11561.602,E2 -11561.602} C_VEL
LIN {X 0,Y 391.919,Z 333.794,A -85,B 0,C 180,E1 -11565.052,E2 -11565.052} C_VEL
LIN {X 0,Y 394.049,Z 343.957,A -85,B 0,C 180,E1 -11568.709,E2 -11568.709} C_VEL
LIN {X 0,Y 394.591,Z 348.094,A -85,B 0,C 180,E1 -11570.121,E2 -11570.121} C_VEL
LIN {X 0,Y 393.757,Z 355.979,A -85,B 0,C 180,E1 -11572.639,E2 -11572.639} C_VEL
LIN {X 0,Y 392.76,Z 366.22,A -85,B 0,C 180,E1 -11575.836,E2 -11575.836} C_VEL
LIN {X 0,Y 391.84,Z 377.932,A -85,B 0,C 180,E1 -11579.42,E2 -11579.42} C_VEL
LIN {X 0,Y 390.891,Z 390.881,A -85,B 0,C 180,E1 -11583.291,E2 -11583.291} C_VEL
LIN {X 0,Y 390.275,Z 402.427,A -85,B 0,C 180,E1 -11586.693,E2 -11586.693} C_VEL
LIN {X 0,Y 390.012,Z 407.394,A -85,B 0,C 180,E1 -11588.079,E2 -11588.079} C_VEL
LIN {X 0,Y 390.407,Z 410.98,A -85,B 0,C 180,E1 -11588.245,E2 -11588.245} C_VEL
LIN {X 0,Y 392.386,Z 426.492,A -85,B 0,C 180,E1 -11588.874,E2 -11588.874} C_VEL
LIN {X 0,Y 393.954,Z 441.065,A -85,B 0,C 180,E1 -11589.662,E2 -11589.662} C_VEL
LIN {X 0,Y 394.692,Z 451.594,A -85,B 0,C 180,E1 -11590.356,E2 -11590.356} C_VEL
LIN {X 0,Y 393.628,Z 465.145,A -85,B 0,C 180,E1 -11591.39,E2 -11591.39} C_VEL
LIN {X 0,Y 392.626,Z 477.436,A -85,B 0,C 180,E1 -11592.554,E2 -11592.554} C_VEL
LIN {X 0,Y 391.522,Z 488.681,A -85,B 0,C 180,E1 -11593.846,E2 -11593.846} C_VEL
LIN {X 0,Y 390.771,Z 498.137,A -85,B 0,C 180,E1 -11595.151,E2 -11595.151} C_VEL
LIN {X 0,Y 390.014,Z 508.365,A -85,B 0,C 180,E1 -11596.842,E2 -11596.842} C_VEL
LIN {X 0,Y 389.579,Z 516.822,A -85,B 0,C 180,E1 -11598.555,E2 -11598.555} C_VEL
LIN {X 0,Y 389.365,Z 523.249,A -85,B 0,C 180,E1 -11600.128,E2 -11600.128} C_VEL
LIN {X 0,Y 389.314,Z 528.501,A -85,B 0,C 180,E1 -11601.697,E2 -11601.697} C_VEL
LIN {X 0,Y 389.346,Z 532.375,A -85,B 0,C 180,E1 -11603.117,E2 -11603.117} C_VEL
LIN {X 0,Y 389.456,Z 536.017,A -85,B 0,C 180,E1 -11604.824,E2 -11604.824} C_VEL
LIN {X 0,Y 389.513,Z 537.683,A -85,B 0,C 180,E1 -11605.862,E2 -11605.862} C_VEL
LIN {X 0,Y 389.571,Z 539.851,A -85,B 0,C 180,E1 -11607.933,E2 -11607.933} C_VEL
LIN {X 0,Y 389.867,Z 540.556,A -85,B 0,C 180,E1 -11610.001,E2 -11610.001} C_VEL
LIN {X 0,Y 389.802,Z 540.318,A -85,B 0,C 180,E1 -11611.034,E2 -11611.034} C_VEL
LIN {X 0,Y 389.566,Z 538.707,A -85,B 0,C 180,E1 -11613.103,E2 -11613.103} C_VEL
LIN {X 0,Y 389.592,Z 537.36,A -85,B 0,C 180,E1 -11614.139,E2 -11614.139} C_VEL
LIN {X 0,Y 389.443,Z 534.582,A -85,B 0,C 180,E1 -11615.697,E2 -11615.697} C_VEL
LIN {X 0,Y 389.339,Z 529.491,A -85,B 0,C 180,E1 -11617.782,E2 -11617.782} C_VEL
LIN {X 0,Y 389.339,Z 522.704,A -85,B 0,C 180,E1 -11619.875,E2 -11619.875} C_VEL
LIN {X 0,Y 389.609,Z 515.231,A -85,B 0,C 180,E1 -11621.709,E2 -11621.709} C_VEL
LIN {X 0,Y 390.168,Z 506.14,A -85,B 0,C 180,E1 -11623.543,E2 -11623.543} C_VEL
LIN {X 0,Y 390.885,Z 496.812,A -85,B 0,C 180,E1 -11625.113,E2 -11625.113} C_VEL
LIN {X 0,Y 391.927,Z 485.788,A -85,B 0,C 180,E1 -11626.674,E2 -11626.674} C_VEL
LIN {X 0,Y 393.231,Z 472.604,A -85,B 0,C 180,E1 -11628.227,E2 -11628.227} C_VEL
LIN {X 0,Y 394.918,Z 458.745,A -85,B 0,C 180,E1 -11629.56,E2 -11629.56} C_VEL
LIN {X 0,Y 395.559,Z 451.888,A -85,B 0,C 180,E1 -11630.136,E2 -11630.136} C_VEL
LIN {X 0,Y 395.387,Z 438.86,A -85,B 0,C 180,E1 -11631.163,E2 -11631.163} C_VEL
LIN {X 0,Y 395,Z 423.959,A -85,B 0,C 180,E1 -11632.154,E2 -11632.154} C_VEL
LIN {X 0,Y 393.37,Z 410.16,A -85,B 0,C 180,E1 -11633.01,E2 -11633.01} C_VEL
LIN {X 0,Y 390.638,Z 396.406,A -85,B 0,C 180,E1 -11633.832,E2 -11633.832} C_VEL
LIN {X 0,Y 389.982,Z 392.858,A -85,B 0,C 180,E1 -11634.073,E2 -11634.073} C_VEL
LIN {X 0,Y 390.058,Z 389.088,A -85,B 0,C 180,E1 -11635.051,E2 -11635.051} C_VEL
LIN {X 0,Y 390.546,Z 376.911,A -85,B 0,C 180,E1 -11638.538,E2 -11638.538} C_VEL
LIN {X 0,Y 391.101,Z 365.754,A -85,B 0,C 180,E1 -11641.902,E2 -11641.902} C_VEL
LIN {X 0,Y 391.99,Z 354.19,A -85,B 0,C 180,E1 -11645.641,E2 -11645.641} C_VEL
LIN {X 0,Y 393.313,Z 345.443,A -85,B 0,C 180,E1 -11648.713,E2 -11648.713} C_VEL
LIN {X 0,Y 393.622,Z 342.482,A -85,B 0,C 180,E1 -11649.848,E2 -11649.848} C_VEL
LIN {X 0,Y 392.793,Z 337.437,A -85,B 0,C 180,E1 -11652.1,E2 -11652.1} C_VEL
LIN {X 0,Y 391.649,Z 331.952,A -85,B 0,C 180,E1 -11654.969,E2 -11654.969} C_VEL
LIN {X 0,Y 390.574,Z 326.834,A -85,B 0,C 180,E1 -11658.258,E2 -11658.258} C_VEL
LIN {X 0,Y 390.087,Z 324.525,A -85,B 0,C 180,E1 -11660.219,E2 -11660.219} C_VEL
LIN {X 0,Y 390.063,Z 324.523,A -85,B 0,C 180,E1 -11663.517,E2 -11663.517} C_VEL
LIN {X 0,Y 390.071,Z 324.521,A -85,B 0,C 180,E1 -11666.046,E2 -11666.046} C_VEL
LIN {X 0,Y 390.05,Z 324.524,A -85,B 0,C 180,E1 -11669.869,E2 -11669.869} C_VEL
LIN {X 0,Y 390.117,Z 324.517,A -85,B 0,C 180,E1 -11673.232,E2 -11673.232} C_VEL
LIN {X 0,Y 390.13,Z 324.7,A -85,B 0,C 180,E1 -11675.523,E2 -11675.523} C_VEL
LIN {X 0,Y 390.486,Z 326.135,A -85,B 0,C 180,E1 -11675.786,E2 -11675.786} C_VEL
LIN {X 0,Y 395.524,Z 336.289,A -85,B 0,C 180,E1 -11676.989,E2 -11676.989} C_VEL
LIN {X 0,Y 399.99,Z 348.075,A -85,B 0,C 180,E1 -11678.348,E2 -11678.348} C_VEL
LIN {X 0,Y 400.617,Z 350.058,A -85,B 0,C 180,E1 -11678.581,E2 -11678.581} C_VEL
LIN {X 0,Y 400.469,Z 354.444,A -85,B 0,C 180,E1 -11678.964,E2 -11678.964} C_VEL
LIN {X 0,Y 399.137,Z 367.356,A -85,B 0,C 180,E1 -11680.187,E2 -11680.187} C_VEL
LIN {X 0,Y 397.871,Z 378.314,A -85,B 0,C 180,E1 -11681.461,E2 -11681.461} C_VEL
LIN {X 0,Y 396.684,Z 387.506,A -85,B 0,C 180,E1 -11682.738,E2 -11682.738} C_VEL
LIN {X 0,Y 395.386,Z 396.502,A -85,B 0,C 180,E1 -11684.224,E2 -11684.224} C_VEL
LIN {X 0,Y 394.262,Z 404.432,A -85,B 0,C 180,E1 -11685.812,E2 -11685.812} C_VEL
LIN {X 0,Y 393.154,Z 411.744,A -85,B 0,C 180,E1 -11687.613,E2 -11687.613} C_VEL
LIN {X 0,Y 392.397,Z 416.84,A -85,B 0,C 180,E1 -11689.161,E2 -11689.161} C_VEL
LIN {X 0,Y 391.607,Z 421.931,A -85,B 0,C 180,E1 -11691.141,E2 -11691.141} C_VEL
LIN {X 0,Y 391.071,Z 425.074,A -85,B 0,C 180,E1 -11692.773,E2 -11692.773} C_VEL
LIN {X 0,Y 390.464,Z 427.76,A -85,B 0,C 180,E1 -11694.837,E2 -11694.837} C_VEL
LIN {X 0,Y 390.246,Z 429.026,A -85,B 0,C 180,E1 -11696.903,E2 -11696.903} C_VEL
LIN {X 0,Y 390.086,Z 428.969,A -85,B 0,C 180,E1 -11698.968,E2 -11698.968} C_VEL
LIN {X 0,Y 389.998,Z 427.58,A -85,B 0,C 180,E1 -11701.033,E2 -11701.033} C_VEL
LIN {X 0,Y 389.907,Z 424.852,A -85,B 0,C 180,E1 -11703.1,E2 -11703.1} C_VEL
LIN {X 0,Y 390.237,Z 420.668,A -85,B 0,C 180,E1 -11705.167,E2 -11705.167} C_VEL
LIN {X 0,Y 390.675,Z 415.398,A -85,B 0,C 180,E1 -11707.073,E2 -11707.073} C_VEL
LIN {X 0,Y 391.179,Z 408.48,A -85,B 0,C 180,E1 -11709.036,E2 -11709.036} C_VEL
LIN {X 0,Y 391.814,Z 400.438,A -85,B 0,C 180,E1 -11710.856,E2 -11710.856} C_VEL
LIN {X 0,Y 392.607,Z 390.611,A -85,B 0,C 180,E1 -11712.667,E2 -11712.667} C_VEL
LIN {X 0,Y 393.42,Z 380.371,A -85,B 0,C 180,E1 -11714.219,E2 -11714.219} C_VEL
LIN {X 0,Y 394.418,Z 368.585,A -85,B 0,C 180,E1 -11715.681,E2 -11715.681} C_VEL
LIN {X 0,Y 395.279,Z 356.394,A -85,B 0,C 180,E1 -11716.927,E2 -11716.927} C_VEL
LIN {X 0,Y 396.019,Z 344.652,A -85,B 0,C 180,E1 -11717.916,E2 -11717.916} C_VEL
LIN {X 0,Y 392.246,Z 331.713,A -85,B 0,C 180,E1 -11719.007,E2 -11719.007} C_VEL
LIN {X 0,Y 390.217,Z 325.145,A -85,B 0,C 180,E1 -11719.532,E2 -11719.532} C_VEL
LIN {X 0,Y 390.116,Z 324.549,A -85,B 0,C 180,E1 -11719.742,E2 -11719.742} C_VEL
LIN {X 0,Y 390.094,Z 324.519,A -85,B 0,C 180,E1 -11723.351,E2 -11723.351} C_VEL
LIN {X 0,Y 390.118,Z 324.517,A -85,B 0,C 180,E1 -11726.768,E2 -11726.768} C_VEL
LIN {X 0,Y 390.044,Z 324.524,A -85,B 0,C 180,E1 -11730.3,E2 -11730.3} C_VEL
LIN {X 0,Y 390.073,Z 324.518,A -85,B 0,C 180,E1 -11734.025,E2 -11734.025} C_VEL
LIN {X 0,Y 390.047,Z 324.52,A -85,B 0,C 180,E1 -11737.551,E2 -11737.551} C_VEL
LIN {X 0,Y 390.061,Z 324.522,A -85,B 0,C 180,E1 -11740.821,E2 -11740.821} C_VEL
LIN {X 0,Y 390.06,Z 324.52,A -85,B 0,C 180,E1 -11743.886,E2 -11743.886} C_VEL
LIN {X 0,Y 390.087,Z 324.516,A -85,B 0,C 180,E1 -11747.619,E2 -11747.619} C_VEL
LIN {X 0,Y 390.098,Z 324.515,A -85,B 0,C 180,E1 -11750.908,E2 -11750.908} C_VEL
LIN {X 0,Y 390.091,Z 324.516,A -85,B 0,C 180,E1 -11754.793,E2 -11754.793} C_VEL
LIN {X 0,Y 390.03,Z 324.526,A -85,B 0,C 180,E1 -11758.495,E2 -11758.495} C_VEL
LIN {X 0,Y 390.123,Z 324.517,A -85,B 0,C 180,E1 -11762.07,E2 -11762.07} C_VEL
LIN {X 0,Y 390.083,Z 324.517,A -85,B 0,C 180,E1 -11765.519,E2 -11765.519} C_VEL
LIN {X 0,Y 390.093,Z 324.516,A -85,B 0,C 180,E1 -11769.529,E2 -11769.529} C_VEL
LIN {X 0,Y 390.144,Z 324.509,A -85,B 0,C 180,E1 -11773.248,E2 -11773.248} C_VEL
LIN {X 0,Y 390.2,Z 324.502,A -85,B 0,C 180,E1 -11776.561,E2 -11776.561} C_VEL
LIN {X 0,Y 390.21,Z 324.5,A -85,B 0,C 180,E1 -11780.67,E2 -11780.67} C_VEL
LIN {X 0,Y 390.323,Z 324.486,A -85,B 0,C 180,E1 -11782.758,E2 -11782.758} C_VEL
LIN {X 0,Y 390.231,Z 324.497,A -85,B 0,C 180,E1 -11784.833,E2 -11784.833} C_VEL
LIN {X 0,Y 390.423,Z 324.478,A -85,B 0,C 180,E1 -11787.936,E2 -11787.936} C_VEL
LIN {X 0,Y 390.553,Z 324.461,A -85,B 0,C 180,E1 -11789.999,E2 -11789.999} C_VEL
LIN {X 0,Y 390.315,Z 324.488,A -85,B 0,C 180,E1 -11793.096,E2 -11793.096} C_VEL
LIN {X 0,Y 390.334,Z 324.486,A -85,B 0,C 180,E1 -11796.201,E2 -11796.201} C_VEL
LIN {X 0,Y 390.318,Z 324.487,A -85,B 0,C 180,E1 -11798.281,E2 -11798.281} C_VEL
LIN {X 0,Y 390.174,Z 324.504,A -85,B 0,C 180,E1 -11802.482,E2 -11802.482} C_VEL
LIN {X 0,Y 390.142,Z 324.513,A -85,B 0,C 180,E1 -11805.676,E2 -11805.676} C_VEL
LIN {X 0,Y 390.108,Z 324.514,A -85,B 0,C 180,E1 -11808.921,E2 -11808.921} C_VEL
LIN {X 0,Y 390.049,Z 324.52,A -85,B 0,C 180,E1 -11812.232,E2 -11812.232} C_VEL
LIN {X 0,Y 390.115,Z 324.514,A -85,B 0,C 180,E1 -11815.819,E2 -11815.819} C_VEL
LIN {X 0,Y 389.408,Z 324.602,A -85,B 0,C 180,E1 -11816.68,E2 -11816.68} C_VEL
LIN {X 0,Y 386.503,Z 324.962,A -85,B 0,C 180,E1 -11818.079,E2 -11818.079} C_VEL
LIN {X 0,Y 384.079,Z 325.269,A -85,B 0,C 180,E1 -11819.21,E2 -11819.21} C_VEL
LIN {X 0,Y 383.066,Z 325.391,A -85,B 0,C 180,E1 -11820.085,E2 -11820.085} C_VEL
LIN {X 0,Y 382.996,Z 325.399,A -85,B 0,C 180,E1 -11820.382,E2 -11820.382} C_VEL
LIN {X 0,Y 383.002,Z 325.403,A -85,B 0,C 180,E1 -11823.399,E2 -11823.399} C_VEL
LIN {X 0,Y 383.03,Z 325.394,A -85,B 0,C 180,E1 -11826.163,E2 -11826.163} C_VEL
LIN {X 0,Y 383.006,Z 325.397,A -85,B 0,C 180,E1 -11829.957,E2 -11829.957} C_VEL
LIN {X 0,Y 383.002,Z 325.401,A -85,B 0,C 180,E1 -11832.777,E2 -11832.777} C_VEL
LIN {X 0,Y 382.997,Z 325.399,A -85,B 0,C 180,E1 -11835.789,E2 -11835.789} C_VEL
LIN {X 0,Y 382.986,Z 325.404,A -85,B 0,C 180,E1 -11838.794,E2 -11838.794} C_VEL
LIN {X 0,Y 382.998,Z 325.398,A -85,B 0,C 180,E1 -11842.095,E2 -11842.095} C_VEL
LIN {X 0,Y 383.013,Z 325.399,A -85,B 0,C 180,E1 -11845.331,E2 -11845.331} C_VEL
LIN {X 0,Y 383.032,Z 325.394,A -85,B 0,C 180,E1 -11847.852,E2 -11847.852} C_VEL
LIN {X 0,Y 383.058,Z 325.391,A -85,B 0,C 180,E1 -11851.719,E2 -11851.719} C_VEL
LIN {X 0,Y 383.046,Z 325.396,A -85,B 0,C 180,E1 -11855.039,E2 -11855.039} C_VEL
LIN {X 0,Y 382.992,Z 325.403,A -85,B 0,C 180,E1 -11858.469,E2 -11858.469} C_VEL
LIN {X 0,Y 383.056,Z 325.391,A -85,B 0,C 180,E1 -11861.826,E2 -11861.826} C_VEL
LIN {X 0,Y 383.103,Z 325.387,A -85,B 0,C 180,E1 -11865.118,E2 -11865.118} C_VEL
LIN {X 0,Y 383.091,Z 325.391,A -85,B 0,C 180,E1 -11868.357,E2 -11868.357} C_VEL
LIN {X 0,Y 383.296,Z 325.362,A -85,B 0,C 180,E1 -11871.932,E2 -11871.932} C_VEL
LIN {X 0,Y 383.193,Z 325.378,A -85,B 0,C 180,E1 -11874.738,E2 -11874.738} C_VEL
LIN {X 0,Y 383.381,Z 325.352,A -85,B 0,C 180,E1 -11877.899,E2 -11877.899} C_VEL
LIN {X 0,Y 383.511,Z 325.337,A -85,B 0,C 180,E1 -11880,E2 -11880} C_VEL
LIN {X 0,Y 383.245,Z 325.368,A -85,B 0,C 180,E1 -11883.153,E2 -11883.153} C_VEL
LIN {X 0,Y 383.279,Z 325.37,A -85,B 0,C 180,E1 -11886.316,E2 -11886.316} C_VEL
LIN {X 0,Y 383.252,Z 325.371,A -85,B 0,C 180,E1 -11888.436,E2 -11888.436} C_VEL
LIN {X 0,Y 383.099,Z 325.387,A -85,B 0,C 180,E1 -11891.642,E2 -11891.642} C_VEL
LIN {X 0,Y 383.107,Z 325.385,A -85,B 0,C 180,E1 -11894.882,E2 -11894.882} C_VEL
LIN {X 0,Y 383.081,Z 325.394,A -85,B 0,C 180,E1 -11898.172,E2 -11898.172} C_VEL
LIN {X 0,Y 382.985,Z 325.401,A -85,B 0,C 180,E1 -11901.531,E2 -11901.531} C_VEL
LIN {X 0,Y 383.044,Z 325.393,A -85,B 0,C 180,E1 -11904.961,E2 -11904.961} C_VEL
LIN {X 0,Y 383.042,Z 325.394,A -85,B 0,C 180,E1 -11908.492,E2 -11908.492} C_VEL
LIN {X 0,Y 383.001,Z 325.399,A -85,B 0,C 180,E1 -11912.428,E2 -11912.428} C_VEL
LIN {X 0,Y 383.027,Z 325.4,A -85,B 0,C 180,E1 -11916.166,E2 -11916.166} C_VEL
LIN {X 0,Y 383.013,Z 325.402,A -85,B 0,C 180,E1 -11919.958,E2 -11919.958} C_VEL
LIN {X 0,Y 383.047,Z 325.499,A -85,B 0,C 180,E1 -11921.216,E2 -11921.216} C_VEL
LIN {X 0,Y 384.938,Z 335.005,A -85,B 0,C 180,E1 -11924.898,E2 -11924.898} C_VEL
LIN {X 0,Y 387.108,Z 345.357,A -85,B 0,C 180,E1 -11928.681,E2 -11928.681} C_VEL
LIN {X 0,Y 387.586,Z 349.499,A -85,B 0,C 180,E1 -11930.122,E2 -11930.122} C_VEL
LIN {X 0,Y 386.783,Z 356.845,A -85,B 0,C 180,E1 -11932.506,E2 -11932.506} C_VEL
LIN {X 0,Y 385.767,Z 366.61,A -85,B 0,C 180,E1 -11935.615,E2 -11935.615} C_VEL
LIN {X 0,Y 384.807,Z 378.235,A -85,B 0,C 180,E1 -11939.245,E2 -11939.245} C_VEL
LIN {X 0,Y 383.911,Z 389.74,A -85,B 0,C 180,E1 -11942.765,E2 -11942.765} C_VEL
LIN {X 0,Y 383.229,Z 402.062,A -85,B 0,C 180,E1 -11946.483,E2 -11946.483} C_VEL
LIN {X 0,Y 382.988,Z 406.62,A -85,B 0,C 180,E1 -11947.762,E2 -11947.762} C_VEL
LIN {X 0,Y 383.534,Z 411.419,A -85,B 0,C 180,E1 -11947.972,E2 -11947.972} C_VEL
LIN {X 0,Y 385.502,Z 427.324,A -85,B 0,C 180,E1 -11948.655,E2 -11948.655} C_VEL
LIN {X 0,Y 386.981,Z 441.555,A -85,B 0,C 180,E1 -11949.462,E2 -11949.462} C_VEL
LIN {X 0,Y 387.654,Z 453.172,A -85,B 0,C 180,E1 -11950.267,E2 -11950.267} C_VEL
LIN {X 0,Y 386.549,Z 466.149,A -85,B 0,C 180,E1 -11951.311,E2 -11951.311} C_VEL
LIN {X 0,Y 385.535,Z 478.075,A -85,B 0,C 180,E1 -11952.497,E2 -11952.497} C_VEL
LIN {X 0,Y 384.427,Z 489.019,A -85,B 0,C 180,E1 -11953.813,E2 -11953.813} C_VEL
LIN {X 0,Y 383.503,Z 499.929,A -85,B 0,C 180,E1 -11955.406,E2 -11955.406} C_VEL
LIN {X 0,Y 382.861,Z 508.937,A -85,B 0,C 180,E1 -11956.994,E2 -11956.994} C_VEL
LIN {X 0,Y 382.503,Z 516.568,A -85,B 0,C 180,E1 -11958.609,E2 -11958.609} C_VEL
LIN {X 0,Y 382.282,Z 523.776,A -85,B 0,C 180,E1 -11960.477,E2 -11960.477} C_VEL
LIN {X 0,Y 382.274,Z 528.762,A -85,B 0,C 180,E1 -11962.076,E2 -11962.076} C_VEL
LIN {X 0,Y 382.302,Z 532.733,A -85,B 0,C 180,E1 -11963.668,E2 -11963.668} C_VEL
LIN {X 0,Y 382.423,Z 534.847,A -85,B 0,C 180,E1 -11964.729,E2 -11964.729} C_VEL
LIN {X 0,Y 382.48,Z 536.535,A -85,B 0,C 180,E1 -11965.786,E2 -11965.786} C_VEL
LIN {X 0,Y 382.546,Z 538.746,A -85,B 0,C 180,E1 -11967.895,E2 -11967.895} C_VEL
LIN {X 0,Y 382.863,Z 539.487,A -85,B 0,C 180,E1 -11970.001,E2 -11970.001} C_VEL
LIN {X 0,Y 382.776,Z 539.258,A -85,B 0,C 180,E1 -11971.053,E2 -11971.053} C_VEL
LIN {X 0,Y 382.527,Z 537.673,A -85,B 0,C 180,E1 -11973.161,E2 -11973.161} C_VEL
LIN {X 0,Y 382.556,Z 536.339,A -85,B 0,C 180,E1 -11974.215,E2 -11974.215} C_VEL
LIN {X 0,Y 382.367,Z 533.584,A -85,B 0,C 180,E1 -11975.803,E2 -11975.803} C_VEL
LIN {X 0,Y 382.252,Z 528.521,A -85,B 0,C 180,E1 -11977.927,E2 -11977.927} C_VEL
LIN {X 0,Y 382.276,Z 521.767,A -85,B 0,C 180,E1 -11980.059,E2 -11980.059} C_VEL
LIN {X 0,Y 382.529,Z 514.345,A -85,B 0,C 180,E1 -11981.929,E2 -11981.929} C_VEL
LIN {X 0,Y 383.17,Z 505.344,A -85,B 0,C 180,E1 -11983.795,E2 -11983.795} C_VEL
LIN {X 0,Y 384.089,Z 494.41,A -85,B 0,C 180,E1 -11985.659,E2 -11985.659} C_VEL
LIN {X 0,Y 385.285,Z 483.229,A -85,B 0,C 180,E1 -11987.243,E2 -11987.243} C_VEL
LIN {X 0,Y 386.646,Z 471.093,A -85,B 0,C 180,E1 -11988.686,E2 -11988.686} C_VEL
LIN {X 0,Y 388.317,Z 457.771,A -85,B 0,C 180,E1 -11989.998,E2 -11989.998} C_VEL
LIN {X 0,Y 388.794,Z 452.027,A -85,B 0,C 180,E1 -11990.502,E2 -11990.502} C_VEL
LIN {X 0,Y 388.805,Z 437.805,A -85,B 0,C 180,E1 -11991.668,E2 -11991.668} C_VEL
LIN {X 0,Y 388.466,Z 423.351,A -85,B 0,C 180,E1 -11992.68,E2 -11992.68} C_VEL
LIN {X 0,Y 386.373,Z 407.034,A -85,B 0,C 180,E1 -11993.754,E2 -11993.754} C_VEL
LIN {X 0,Y 383.689,Z 394.535,A -85,B 0,C 180,E1 -11994.571,E2 -11994.571} C_VEL
LIN {X 0,Y 382.968,Z 390.821,A -85,B 0,C 180,E1 -11994.85,E2 -11994.85} C_VEL
LIN {X 0,Y 383.378,Z 380.356,A -85,B 0,C 180,E1 -11997.837,E2 -11997.837} C_VEL
LIN {X 0,Y 383.915,Z 370.49,A -85,B 0,C 180,E1 -12000.836,E2 -12000.836} C_VEL
LIN {X 0,Y 384.665,Z 359.177,A -85,B 0,C 180,E1 -12004.499,E2 -12004.499} C_VEL
LIN {X 0,Y 386.157,Z 348.549,A -85,B 0,C 180,E1 -12008.229,E2 -12008.229} C_VEL
LIN {X 0,Y 386.754,Z 345.198,A -85,B 0,C 180,E1 -12009.496,E2 -12009.496} C_VEL
LIN {X 0,Y 386.412,Z 341.952,A -85,B 0,C 180,E1 -12010.902,E2 -12010.902} C_VEL
LIN {X 0,Y 385.523,Z 337.258,A -85,B 0,C 180,E1 -12013.182,E2 -12013.182} C_VEL
LIN {X 0,Y 384.478,Z 332.297,A -85,B 0,C 180,E1 -12016.004,E2 -12016.004} C_VEL
LIN {X 0,Y 383.656,Z 328.311,A -85,B 0,C 180,E1 -12018.741,E2 -12018.741} C_VEL
LIN {X 0,Y 383.055,Z 325.474,A -85,B 0,C 180,E1 -12021.144,E2 -12021.144} C_VEL
LIN {X 0,Y 383.03,Z 325.399,A -85,B 0,C 180,E1 -12024.045,E2 -12024.045} C_VEL
LIN {X 0,Y 382.99,Z 325.404,A -85,B 0,C 180,E1 -12027.578,E2 -12027.578} C_VEL
LIN {X 0,Y 382.995,Z 325.402,A -85,B 0,C 180,E1 -12030.301,E2 -12030.301} C_VEL
LIN {X 0,Y 383.084,Z 325.392,A -85,B 0,C 180,E1 -12034.021,E2 -12034.021} C_VEL
LIN {X 0,Y 383.119,Z 325.674,A -85,B 0,C 180,E1 -12034.754,E2 -12034.754} C_VEL
LIN {X 0,Y 383.615,Z 327.339,A -85,B 0,C 180,E1 -12035.041,E2 -12035.041} C_VEL
LIN {X 0,Y 386.949,Z 333.494,A -85,B 0,C 180,E1 -12035.841,E2 -12035.841} C_VEL
LIN {X 0,Y 391.696,Z 344.466,A -85,B 0,C 180,E1 -12037.194,E2 -12037.194} C_VEL
LIN {X 0,Y 394.432,Z 352.525,A -85,B 0,C 180,E1 -12038.184,E2 -12038.184} C_VEL
LIN {X 0,Y 394.354,Z 355.871,A -85,B 0,C 180,E1 -12038.493,E2 -12038.493} C_VEL
LIN {X 0,Y 392.918,Z 368.59,A -85,B 0,C 180,E1 -12039.724,E2 -12039.724} C_VEL
LIN {X 0,Y 391.573,Z 379.478,A -85,B 0,C 180,E1 -12041.016,E2 -12041.016} C_VEL
LIN {X 0,Y 390.1,Z 389.956,A -85,B 0,C 180,E1 -12042.511,E2 -12042.511} C_VEL
LIN {X 0,Y 388.846,Z 397.944,A -85,B 0,C 180,E1 -12043.878,E2 -12043.878} C_VEL
LIN {X 0,Y 387.596,Z 406.108,A -85,B 0,C 180,E1 -12045.563,E2 -12045.563} C_VEL
LIN {X 0,Y 386.412,Z 413.3,A -85,B 0,C 180,E1 -12047.394,E2 -12047.394} C_VEL
LIN {X 0,Y 385.587,Z 418.317,A -85,B 0,C 180,E1 -12048.967,E2 -12048.967} C_VEL
LIN {X 0,Y 384.787,Z 423.114,A -85,B 0,C 180,E1 -12050.887,E2 -12050.887} C_VEL
LIN {X 0,Y 384.148,Z 426.396,A -85,B 0,C 180,E1 -12052.642,E2 -12052.642} C_VEL
LIN {X 0,Y 383.51,Z 428.988,A -85,B 0,C 180,E1 -12054.743,E2 -12054.743} C_VEL
LIN {X 0,Y 383.264,Z 430.177,A -85,B 0,C 180,E1 -12056.847,E2 -12056.847} C_VEL
LIN {X 0,Y 383.073,Z 430.047,A -85,B 0,C 180,E1 -12058.949,E2 -12058.949} C_VEL
LIN {X 0,Y 382.991,Z 428.585,A -85,B 0,C 180,E1 -12061.052,E2 -12061.052} C_VEL
LIN {X 0,Y 382.879,Z 425.782,A -85,B 0,C 180,E1 -12063.157,E2 -12063.157} C_VEL
LIN {X 0,Y 383.228,Z 421.515,A -85,B 0,C 180,E1 -12065.261,E2 -12065.261} C_VEL
LIN {X 0,Y 383.666,Z 416.423,A -85,B 0,C 180,E1 -12067.112,E2 -12067.112} C_VEL
LIN {X 0,Y 384.105,Z 410.452,A -85,B 0,C 180,E1 -12068.866,E2 -12068.866} C_VEL
LIN {X 0,Y 384.773,Z 402.267,A -85,B 0,C 180,E1 -12070.791,E2 -12070.791} C_VEL
LIN {X 0,Y 385.384,Z 394.109,A -85,B 0,C 180,E1 -12072.373,E2 -12072.373} C_VEL
LIN {X 0,Y 386.199,Z 384.325,A -85,B 0,C 180,E1 -12073.953,E2 -12073.953} C_VEL
LIN {X 0,Y 387.183,Z 373.564,A -85,B 0,C 180,E1 -12075.395,E2 -12075.395} C_VEL
LIN {X 0,Y 388.096,Z 361.905,A -85,B 0,C 180,E1 -12076.696,E2 -12076.696} C_VEL
LIN {X 0,Y 388.897,Z 350.46,A -85,B 0,C 180,E1 -12077.756,E2 -12077.756} C_VEL
LIN {X 0,Y 389.153,Z 347.07,A -85,B 0,C 180,E1 -12078.034,E2 -12078.034} C_VEL
LIN {X 0,Y 387.72,Z 341.09,A -85,B 0,C 180,E1 -12078.57,E2 -12078.57} C_VEL
LIN {X 0,Y 383.188,Z 325.989,A -85,B 0,C 180,E1 -12079.818,E2 -12079.818} C_VEL
LIN {X 0,Y 383.081,Z 325.449,A -85,B 0,C 180,E1 -12079.98,E2 -12079.98} C_VEL
LIN {X 0,Y 383.039,Z 325.397,A -85,B 0,C 180,E1 -12083.807,E2 -12083.807} C_VEL
LIN {X 0,Y 383.062,Z 325.391,A -85,B 0,C 180,E1 -12087.302,E2 -12087.302} C_VEL
LIN {X 0,Y 382.988,Z 325.403,A -85,B 0,C 180,E1 -12090.919,E2 -12090.919} C_VEL
LIN {X 0,Y 383.023,Z 325.401,A -85,B 0,C 180,E1 -12094.668,E2 -12094.668} C_VEL
LIN {X 0,Y 383.003,Z 325.399,A -85,B 0,C 180,E1 -12097.903,E2 -12097.903} C_VEL
LIN {X 0,Y 382.989,Z 325.4,A -85,B 0,C 180,E1 -12101.347,E2 -12101.347} C_VEL
LIN {X 0,Y 383.002,Z 325.403,A -85,B 0,C 180,E1 -12104.303,E2 -12104.303} C_VEL
LIN {X 0,Y 383.045,Z 325.393,A -85,B 0,C 180,E1 -12107.244,E2 -12107.244} C_VEL
LIN {X 0,Y 383.025,Z 325.401,A -85,B 0,C 180,E1 -12110.413,E2 -12110.413} C_VEL
LIN {X 0,Y 383.031,Z 325.398,A -85,B 0,C 180,E1 -12114.044,E2 -12114.044} C_VEL
LIN {X 0,Y 382.993,Z 325.4,A -85,B 0,C 180,E1 -12117.578,E2 -12117.578} C_VEL
LIN {X 0,Y 382.998,Z 325.404,A -85,B 0,C 180,E1 -12120.3,E2 -12120.3} C_VEL
LIN {X 0,Y 383.086,Z 325.393,A -85,B 0,C 180,E1 -12124.02,E2 -12124.02} C_VEL
LIN {X 0,Y 382.997,Z 325.399,A -85,B 0,C 180,E1 -12127.334,E2 -12127.334} C_VEL
LIN {X 0,Y 383.067,Z 325.39,A -85,B 0,C 180,E1 -12130.716,E2 -12130.716} C_VEL
LIN {X 0,Y 383.087,Z 325.394,A -85,B 0,C 180,E1 -12134.026,E2 -12134.026} C_VEL
LIN {X 0,Y 383.142,Z 325.381,A -85,B 0,C 180,E1 -12137.283,E2 -12137.283} C_VEL
LIN {X 0,Y 383.157,Z 325.38,A -85,B 0,C 180,E1 -12140.497,E2 -12140.497} C_VEL
LIN {X 0,Y 383.278,Z 325.364,A -85,B 0,C 180,E1 -12142.624,E2 -12142.624} C_VEL
LIN {X 0,Y 383.203,Z 325.373,A -85,B 0,C 180,E1 -12144.738,E2 -12144.738} C_VEL
LIN {X 0,Y 383.39,Z 325.355,A -85,B 0,C 180,E1 -12147.898,E2 -12147.898} C_VEL
LIN {X 0,Y 383.523,Z 325.337,A -85,B 0,C 180,E1 -12149.999,E2 -12149.999} C_VEL
LIN {X 0,Y 383.252,Z 325.368,A -85,B 0,C 180,E1 -12153.153,E2 -12153.153} C_VEL
LIN {X 0,Y 383.291,Z 325.363,A -85,B 0,C 180,E1 -12156.315,E2 -12156.315} C_VEL
LIN {X 0,Y 383.264,Z 325.365,A -85,B 0,C 180,E1 -12158.435,E2 -12158.435} C_VEL
LIN {X 0,Y 383.102,Z 325.391,A -85,B 0,C 180,E1 -12161.641,E2 -12161.641} C_VEL
LIN {X 0,Y 383.113,Z 325.385,A -85,B 0,C 180,E1 -12164.88,E2 -12164.88} C_VEL
LIN {X 0,Y 383.065,Z 325.391,A -85,B 0,C 180,E1 -12168.172,E2 -12168.172} C_VEL
LIN {X 0,Y 383.001,Z 325.404,A -85,B 0,C 180,E1 -12171.529,E2 -12171.529} C_VEL
LIN {X 0,Y 383.053,Z 325.394,A -85,B 0,C 180,E1 -12174.959,E2 -12174.959} C_VEL
LIN {X 0,Y 383.03,Z 325.394,A -85,B 0,C 180,E1 -12178.269,E2 -12178.269} C_VEL
LIN {X 0,Y 382.996,Z 325.399,A -85,B 0,C 180,E1 -12180.382,E2 -12180.382} C_VEL
LIN {X 0,Y 382.367,Z 325.484,A -85,B 0,C 180,E1 -12181.258,E2 -12181.258} C_VEL
LIN {X 0,Y 379.532,Z 325.831,A -85,B 0,C 180,E1 -12182.684,E2 -12182.684} C_VEL
LIN {X 0,Y 377.103,Z 326.134,A -85,B 0,C 180,E1 -12183.836,E2 -12183.836} C_VEL
LIN {X 0,Y 376.05,Z 326.266,A -85,B 0,C 180,E1 -12184.728,E2 -12184.728} C_VEL
LIN {X 0,Y 375.959,Z 326.277,A -85,B 0,C 180,E1 -12185.03,E2 -12185.03} C_VEL
LIN {X 0,Y 375.972,Z 326.274,A -85,B 0,C 180,E1 -12188.269,E2 -12188.269} C_VEL
LIN {X 0,Y 375.933,Z 326.28,A -85,B 0,C 180,E1 -12191.6,E2 -12191.6} C_VEL
LIN {X 0,Y 375.952,Z 326.28,A -85,B 0,C 180,E1 -12195.263,E2 -12195.263} C_VEL
LIN {X 0,Y 375.937,Z 326.283,A -85,B 0,C 180,E1 -12199.132,E2 -12199.132} C_VEL
LIN {X 0,Y 375.962,Z 326.275,A -85,B 0,C 180,E1 -12201.911,E2 -12201.911} C_VEL
LIN {X 0,Y 375.975,Z 326.275,A -85,B 0,C 180,E1 -12205.331,E2 -12205.331} C_VEL
LIN {X 0,Y 375.972,Z 326.276,A -85,B 0,C 180,E1 -12208.439,E2 -12208.439} C_VEL
LIN {X 0,Y 375.996,Z 326.271,A -85,B 0,C 180,E1 -12212.141,E2 -12212.141} C_VEL
LIN {X 0,Y 376,Z 326.274,A -85,B 0,C 180,E1 -12214.538,E2 -12214.538} C_VEL
LIN {X 0,Y 375.961,Z 326.276,A -85,B 0,C 180,E1 -12218.045,E2 -12218.045} C_VEL
LIN {X 0,Y 376.002,Z 326.27,A -85,B 0,C 180,E1 -12221.472,E2 -12221.472} C_VEL
LIN {X 0,Y 376.051,Z 326.268,A -85,B 0,C 180,E1 -12224.832,E2 -12224.832} C_VEL
LIN {X 0,Y 376.043,Z 326.267,A -85,B 0,C 180,E1 -12228.136,E2 -12228.136} C_VEL
LIN {X 0,Y 376.25,Z 326.24,A -85,B 0,C 180,E1 -12231.877,E2 -12231.877} C_VEL
LIN {X 0,Y 376.165,Z 326.254,A -85,B 0,C 180,E1 -12234.64,E2 -12234.64} C_VEL
LIN {X 0,Y 376.347,Z 326.228,A -85,B 0,C 180,E1 -12237.859,E2 -12237.859} C_VEL
LIN {X 0,Y 376.481,Z 326.213,A -85,B 0,C 180,E1 -12240,E2 -12240} C_VEL
LIN {X 0,Y 376.183,Z 326.247,A -85,B 0,C 180,E1 -12243.213,E2 -12243.213} C_VEL
LIN {X 0,Y 376.239,Z 326.245,A -85,B 0,C 180,E1 -12246.435,E2 -12246.435} C_VEL
LIN {X 0,Y 376.198,Z 326.248,A -85,B 0,C 180,E1 -12248.595,E2 -12248.595} C_VEL
LIN {X 0,Y 376.051,Z 326.267,A -85,B 0,C 180,E1 -12251.863,E2 -12251.863} C_VEL
LIN {X 0,Y 376.054,Z 326.263,A -85,B 0,C 180,E1 -12255.167,E2 -12255.167} C_VEL
LIN {X 0,Y 376.016,Z 326.27,A -85,B 0,C 180,E1 -12258.526,E2 -12258.526} C_VEL
LIN {X 0,Y 375.955,Z 326.281,A -85,B 0,C 180,E1 -12261.955,E2 -12261.955} C_VEL
LIN {X 0,Y 375.998,Z 326.272,A -85,B 0,C 180,E1 -12265.461,E2 -12265.461} C_VEL
LIN {X 0,Y 375.969,Z 326.274,A -85,B 0,C 180,E1 -12269.079,E2 -12269.079} C_VEL
LIN {X 0,Y 375.951,Z 326.276,A -85,B 0,C 180,E1 -12272.828,E2 -12272.828} C_VEL
LIN {X 0,Y 375.951,Z 326.278,A -85,B 0,C 180,E1 -12275.416,E2 -12275.416} C_VEL
LIN {X 0,Y 375.971,Z 326.279,A -85,B 0,C 180,E1 -12278.272,E2 -12278.272} C_VEL
LIN {X 0,Y 376.002,Z 326.365,A -85,B 0,C 180,E1 -12280.859,E2 -12280.859} C_VEL
LIN {X 0,Y 377.667,Z 334.947,A -85,B 0,C 180,E1 -12284.254,E2 -12284.254} C_VEL
LIN {X 0,Y 379.618,Z 344.313,A -85,B 0,C 180,E1 -12287.777,E2 -12287.777} C_VEL
LIN {X 0,Y 380.563,Z 349.755,A -85,B 0,C 180,E1 -12289.734,E2 -12289.734} C_VEL
LIN {X 0,Y 380.314,Z 353.741,A -85,B 0,C 180,E1 -12291.077,E2 -12291.077} C_VEL
LIN {X 0,Y 378.963,Z 365.472,A -85,B 0,C 180,E1 -12294.909,E2 -12294.909} C_VEL
LIN {X 0,Y 377.833,Z 377.741,A -85,B 0,C 180,E1 -12298.83,E2 -12298.83} C_VEL
LIN {X 0,Y 376.953,Z 388.58,A -85,B 0,C 180,E1 -12302.22,E2 -12302.22} C_VEL
LIN {X 0,Y 376.287,Z 399.981,A -85,B 0,C 180,E1 -12305.74,E2 -12305.74} C_VEL
LIN {X 0,Y 375.95,Z 405.727,A -85,B 0,C 180,E1 -12307.431,E2 -12307.431} C_VEL
LIN {X 0,Y 376.795,Z 413.039,A -85,B 0,C 180,E1 -12307.746,E2 -12307.746} C_VEL
LIN {X 0,Y 378.545,Z 427.669,A -85,B 0,C 180,E1 -12308.411,E2 -12308.411} C_VEL
LIN {X 0,Y 380.076,Z 442.985,A -85,B 0,C 180,E1 -12309.329,E2 -12309.329} C_VEL
LIN {X 0,Y 380.687,Z 453.453,A -85,B 0,C 180,E1 -12310.087,E2 -12310.087} C_VEL
LIN {X 0,Y 379.488,Z 467.022,A -85,B 0,C 180,E1 -12311.235,E2 -12311.235} C_VEL
LIN {X 0,Y 378.295,Z 479.694,A -85,B 0,C 180,E1 -12312.569,E2 -12312.569} C_VEL
LIN {X 0,Y 377.179,Z 491.193,A -85,B 0,C 180,E1 -12314.049,E2 -12314.049} C_VEL
LIN {X 0,Y 376.283,Z 501.591,A -85,B 0,C 180,E1 -12315.673,E2 -12315.673} C_VEL
LIN {X 0,Y 375.701,Z 510.226,A -85,B 0,C 180,E1 -12317.304,E2 -12317.304} C_VEL
LIN {X 0,Y 375.352,Z 518.482,A -85,B 0,C 180,E1 -12319.209,E2 -12319.209} C_VEL
LIN {X 0,Y 375.207,Z 524.259,A -85,B 0,C 180,E1 -12320.84,E2 -12320.84} C_VEL
LIN {X 0,Y 375.249,Z 528.922,A -85,B 0,C 180,E1 -12322.468,E2 -12322.468} C_VEL
LIN {X 0,Y 375.39,Z 533.648,A -85,B 0,C 180,E1 -12324.63,E2 -12324.63} C_VEL
LIN {X 0,Y 375.448,Z 535.373,A -85,B 0,C 180,E1 -12325.707,E2 -12325.707} C_VEL
LIN {X 0,Y 375.522,Z 537.627,A -85,B 0,C 180,E1 -12327.856,E2 -12327.856} C_VEL
LIN {X 0,Y 375.857,Z 538.411,A -85,B 0,C 180,E1 -12330.001,E2 -12330.001} C_VEL
LIN {X 0,Y 375.749,Z 538.197,A -85,B 0,C 180,E1 -12331.073,E2 -12331.073} C_VEL
LIN {X 0,Y 375.489,Z 536.638,A -85,B 0,C 180,E1 -12333.22,E2 -12333.22} C_VEL
LIN {X 0,Y 375.517,Z 535.322,A -85,B 0,C 180,E1 -12334.294,E2 -12334.294} C_VEL
LIN {X 0,Y 375.278,Z 531.486,A -85,B 0,C 180,E1 -12336.453,E2 -12336.453} C_VEL
LIN {X 0,Y 375.156,Z 526.072,A -85,B 0,C 180,E1 -12338.62,E2 -12338.62} C_VEL
LIN {X 0,Y 375.201,Z 520.856,A -85,B 0,C 180,E1 -12340.251,E2 -12340.251} C_VEL
LIN {X 0,Y 375.487,Z 513.504,A -85,B 0,C 180,E1 -12342.156,E2 -12342.156} C_VEL
LIN {X 0,Y 376.165,Z 504.584,A -85,B 0,C 180,E1 -12344.058,E2 -12344.058} C_VEL
LIN {X 0,Y 377.168,Z 493.825,A -85,B 0,C 180,E1 -12345.954,E2 -12345.954} C_VEL
LIN {X 0,Y 378.436,Z 482.808,A -85,B 0,C 180,E1 -12347.565,E2 -12347.565} C_VEL
LIN {X 0,Y 380.075,Z 469.708,A -85,B 0,C 180,E1 -12349.161,E2 -12349.161} C_VEL
LIN {X 0,Y 382.001,Z 455.299,A -85,B 0,C 180,E1 -12350.602,E2 -12350.602} C_VEL
LIN {X 0,Y 382.22,Z 439.935,A -85,B 0,C 180,E1 -12351.954,E2 -12351.954} C_VEL
LIN {X 0,Y 382.157,Z 426.455,A -85,B 0,C 180,E1 -12352.968,E2 -12352.968} C_VEL
LIN {X 0,Y 380.802,Z 412.652,A -85,B 0,C 180,E1 -12353.956,E2 -12353.956} C_VEL
LIN {X 0,Y 378.125,Z 397.963,A -85,B 0,C 180,E1 -12354.985,E2 -12354.985} C_VEL
LIN {X 0,Y 376.048,Z 389.184,A -85,B 0,C 180,E1 -12355.635,E2 -12355.635} C_VEL
LIN {X 0,Y 376.052,Z 387.761,A -85,B 0,C 180,E1 -12355.93,E2 -12355.93} C_VEL
LIN {X 0,Y 376.694,Z 375.582,A -85,B 0,C 180,E1 -12359.632,E2 -12359.632} C_VEL
LIN {X 0,Y 377.464,Z 363.83,A -85,B 0,C 180,E1 -12363.44,E2 -12363.44} C_VEL
LIN {X 0,Y 378.998,Z 351.663,A -85,B 0,C 180,E1 -12367.731,E2 -12367.731} C_VEL
LIN {X 0,Y 379.881,Z 346.654,A -85,B 0,C 180,E1 -12369.664,E2 -12369.664} C_VEL
LIN {X 0,Y 379.249,Z 341.875,A -85,B 0,C 180,E1 -12371.847,E2 -12371.847} C_VEL
LIN {X 0,Y 378.03,Z 335.928,A -85,B 0,C 180,E1 -12375.052,E2 -12375.052} C_VEL
LIN {X 0,Y 377.015,Z 331.148,A -85,B 0,C 180,E1 -12378.216,E2 -12378.216} C_VEL
LIN {X 0,Y 376.404,Z 328.229,A -85,B 0,C 180,E1 -12380.593,E2 -12380.593} C_VEL
LIN {X 0,Y 375.957,Z 326.297,A -85,B 0,C 180,E1 -12382.588,E2 -12382.588} C_VEL
LIN {X 0,Y 375.963,Z 326.278,A -85,B 0,C 180,E1 -12385.889,E2 -12385.889} C_VEL
LIN {X 0,Y 375.968,Z 326.279,A -85,B 0,C 180,E1 -12389.688,E2 -12389.688} C_VEL
LIN {X 0,Y 376.023,Z 326.273,A -85,B 0,C 180,E1 -12393.348,E2 -12393.348} C_VEL
LIN {X 0,Y 376.094,Z 326.603,A -85,B 0,C 180,E1 -12393.893,E2 -12393.893} C_VEL
LIN {X 0,Y 376.496,Z 327.986,A -85,B 0,C 180,E1 -12394.138,E2 -12394.138} C_VEL
LIN {X 0,Y 380.66,Z 335.62,A -85,B 0,C 180,E1 -12395.215,E2 -12395.215} C_VEL
LIN {X 0,Y 384.967,Z 345.228,A -85,B 0,C 180,E1 -12396.495,E2 -12396.495} C_VEL
LIN {X 0,Y 388.386,Z 355.337,A -85,B 0,C 180,E1 -12397.802,E2 -12397.802} C_VEL
LIN {X 0,Y 387.109,Z 367.553,A -85,B 0,C 180,E1 -12398.988,E2 -12398.988} C_VEL
LIN {X 0,Y 385.734,Z 377.752,A -85,B 0,C 180,E1 -12400.163,E2 -12400.163} C_VEL
LIN {X 0,Y 384.211,Z 388.169,A -85,B 0,C 180,E1 -12401.607,E2 -12401.607} C_VEL
LIN {X 0,Y 382.653,Z 397.798,A -85,B 0,C 180,E1 -12403.22,E2 -12403.22} C_VEL
LIN {X 0,Y 381.571,Z 404.294,A -85,B 0,C 180,E1 -12404.51,E2 -12404.51} C_VEL
LIN {X 0,Y 380.429,Z 411.05,A -85,B 0,C 180,E1 -12406.104,E2 -12406.104} C_VEL
LIN {X 0,Y 379.398,Z 416.668,A -85,B 0,C 180,E1 -12407.7,E2 -12407.7} C_VEL
LIN {X 0,Y 378.567,Z 421.222,A -85,B 0,C 180,E1 -12409.301,E2 -12409.301} C_VEL
LIN {X 0,Y 377.617,Z 425.95,A -85,B 0,C 180,E1 -12411.438,E2 -12411.438} C_VEL
LIN {X 0,Y 376.828,Z 429.161,A -85,B 0,C 180,E1 -12413.575,E2 -12413.575} C_VEL
LIN {X 0,Y 376.389,Z 430.951,A -85,B 0,C 180,E1 -12415.717,E2 -12415.717} C_VEL
LIN {X 0,Y 376.164,Z 431.398,A -85,B 0,C 180,E1 -12417.859,E2 -12417.859} C_VEL
LIN {X 0,Y 376.005,Z 430.527,A -85,B 0,C 180,E1 -12420,E2 -12420} C_VEL
LIN {X 0,Y 375.952,Z 428.31,A -85,B 0,C 180,E1 -12422.143,E2 -12422.143} C_VEL
LIN {X 0,Y 375.983,Z 424.714,A -85,B 0,C 180,E1 -12424.288,E2 -12424.288} C_VEL
LIN {X 0,Y 376.497,Z 419.55,A -85,B 0,C 180,E1 -12426.431,E2 -12426.431} C_VEL
LIN {X 0,Y 376.915,Z 414.625,A -85,B 0,C 180,E1 -12428.039,E2 -12428.039} C_VEL
LIN {X 0,Y 377.399,Z 407.569,A -85,B 0,C 180,E1 -12429.919,E2 -12429.919} C_VEL
LIN {X 0,Y 378.186,Z 398.835,A -85,B 0,C 180,E1 -12431.796,E2 -12431.796} C_VEL
LIN {X 0,Y 378.928,Z 389.796,A -85,B 0,C 180,E1 -12433.406,E2 -12433.406} C_VEL
LIN {X 0,Y 379.71,Z 380.903,A -85,B 0,C 180,E1 -12434.744,E2 -12434.744} C_VEL
LIN {X 0,Y 380.608,Z 370.401,A -85,B 0,C 180,E1 -12436.08,E2 -12436.08} C_VEL
LIN {X 0,Y 381.563,Z 357.731,A -85,B 0,C 180,E1 -12437.416,E2 -12437.416} C_VEL
LIN {X 0,Y 382.264,Z 348.754,A -85,B 0,C 180,E1 -12438.213,E2 -12438.213} C_VEL
LIN {X 0,Y 381.654,Z 345.572,A -85,B 0,C 180,E1 -12438.501,E2 -12438.501} C_VEL
LIN {X 0,Y 377.574,Z 331.67,A -85,B 0,C 180,E1 -12439.699,E2 -12439.699} C_VEL
LIN {X 0,Y 376.137,Z 326.779,A -85,B 0,C 180,E1 -12440.116,E2 -12440.116} C_VEL
LIN {X 0,Y 376.018,Z 326.287,A -85,B 0,C 180,E1 -12440.372,E2 -12440.372} C_VEL
LIN {X 0,Y 375.999,Z 326.276,A -85,B 0,C 180,E1 -12444.282,E2 -12444.282} C_VEL
LIN {X 0,Y 376.025,Z 326.273,A -85,B 0,C 180,E1 -12446.652,E2 -12446.652} C_VEL
LIN {X 0,Y 375.975,Z 326.275,A -85,B 0,C 180,E1 -12449.079,E2 -12449.079} C_VEL
LIN {X 0,Y 375.954,Z 326.28,A -85,B 0,C 180,E1 -12452.829,E2 -12452.829} C_VEL
LIN {X 0,Y 375.963,Z 326.275,A -85,B 0,C 180,E1 -12455.415,E2 -12455.415} C_VEL
LIN {X 0,Y 375.978,Z 326.277,A -85,B 0,C 180,E1 -12458.27,E2 -12458.27} C_VEL
LIN {X 0,Y 375.939,Z 326.278,A -85,B 0,C 180,E1 -12461.601,E2 -12461.601} C_VEL
LIN {X 0,Y 375.934,Z 326.278,A -85,B 0,C 180,E1 -12465.268,E2 -12465.268} C_VEL
LIN {X 0,Y 375.965,Z 326.281,A -85,B 0,C 180,E1 -12468.395,E2 -12468.395} C_VEL
LIN {X 0,Y 375.981,Z 326.274,A -85,B 0,C 180,E1 -12471.729,E2 -12471.729} C_VEL
LIN {X 0,Y 375.986,Z 326.272,A -85,B 0,C 180,E1 -12475.332,E2 -12475.332} C_VEL
LIN {X 0,Y 375.964,Z 326.279,A -85,B 0,C 180,E1 -12478.438,E2 -12478.438} C_VEL
LIN {X 0,Y 375.99,Z 326.278,A -85,B 0,C 180,E1 -12482.14,E2 -12482.14} C_VEL
LIN {X 0,Y 376.011,Z 326.271,A -85,B 0,C 180,E1 -12484.538,E2 -12484.538} C_VEL
LIN {X 0,Y 375.962,Z 326.281,A -85,B 0,C 180,E1 -12488.045,E2 -12488.045} C_VEL
LIN {X 0,Y 376.03,Z 326.268,A -85,B 0,C 180,E1 -12491.473,E2 -12491.473} C_VEL
LIN {X 0,Y 376.064,Z 326.262,A -85,B 0,C 180,E1 -12494.832,E2 -12494.832} C_VEL
LIN {X 0,Y 376.056,Z 326.267,A -85,B 0,C 180,E1 -12498.136,E2 -12498.136} C_VEL
LIN {X 0,Y 376.263,Z 326.244,A -85,B 0,C 180,E1 -12501.877,E2 -12501.877} C_VEL
LIN {X 0,Y 376.175,Z 326.248,A -85,B 0,C 180,E1 -12504.639,E2 -12504.639} C_VEL
LIN {X 0,Y 376.356,Z 326.231,A -85,B 0,C 180,E1 -12507.859,E2 -12507.859} C_VEL
LIN {X 0,Y 376.492,Z 326.213,A -85,B 0,C 180,E1 -12509.999,E2 -12509.999} C_VEL
LIN {X 0,Y 376.19,Z 326.248,A -85,B 0,C 180,E1 -12513.212,E2 -12513.212} C_VEL
LIN {X 0,Y 376.251,Z 326.239,A -85,B 0,C 180,E1 -12516.434,E2 -12516.434} C_VEL
LIN {X 0,Y 376.209,Z 326.244,A -85,B 0,C 180,E1 -12518.594,E2 -12518.594} C_VEL
LIN {X 0,Y 376.054,Z 326.267,A -85,B 0,C 180,E1 -12521.862,E2 -12521.862} C_VEL
LIN {X 0,Y 376.061,Z 326.265,A -85,B 0,C 180,E1 -12525.166,E2 -12525.166} C_VEL
LIN {X 0,Y 376.011,Z 326.269,A -85,B 0,C 180,E1 -12528.525,E2 -12528.525} C_VEL
LIN {X 0,Y 375.969,Z 326.275,A -85,B 0,C 180,E1 -12531.953,E2 -12531.953} C_VEL
LIN {X 0,Y 376.008,Z 326.275,A -85,B 0,C 180,E1 -12535.46,E2 -12535.46} C_VEL
LIN {X 0,Y 375.961,Z 326.279,A -85,B 0,C 180,E1 -12539.079,E2 -12539.079} C_VEL
LIN {X 0,Y 375.948,Z 326.279,A -85,B 0,C 180,E1 -12542.827,E2 -12542.827} C_VEL
LIN {X 0,Y 375.959,Z 326.277,A -85,B 0,C 180,E1 -12545.03,E2 -12545.03} C_VEL
LIN {X 0,Y 375.274,Z 326.365,A -85,B 0,C 180,E1 -12545.924,E2 -12545.924} C_VEL
LIN {X 0,Y 372.398,Z 326.723,A -85,B 0,C 180,E1 -12547.376,E2 -12547.376} C_VEL
LIN {X 0,Y 369.979,Z 327.021,A -85,B 0,C 180,E1 -12548.551,E2 -12548.551} C_VEL
LIN {X 0,Y 368.955,Z 327.151,A -85,B 0,C 180,E1 -12549.46,E2 -12549.46} C_VEL
LIN {X 0,Y 368.879,Z 327.156,A -85,B 0,C 180,E1 -12549.768,E2 -12549.768} C_VEL
LIN {X 0,Y 368.884,Z 327.161,A -85,B 0,C 180,E1 -12553.303,E2 -12553.303} C_VEL
LIN {X 0,Y 368.883,Z 327.16,A -85,B 0,C 180,E1 -12556.695,E2 -12556.695} C_VEL
LIN {X 0,Y 368.909,Z 327.154,A -85,B 0,C 180,E1 -12559.642,E2 -12559.642} C_VEL
LIN {X 0,Y 368.899,Z 327.159,A -85,B 0,C 180,E1 -12563.143,E2 -12563.143} C_VEL
LIN {X 0,Y 368.896,Z 327.157,A -85,B 0,C 180,E1 -12566.461,E2 -12566.461} C_VEL
LIN {X 0,Y 368.919,Z 327.154,A -85,B 0,C 180,E1 -12570.31,E2 -12570.31} C_VEL
LIN {X 0,Y 368.976,Z 327.146,A -85,B 0,C 180,E1 -12573.534,E2 -12573.534} C_VEL
LIN {X 0,Y 368.96,Z 327.15,A -85,B 0,C 180,E1 -12576.421,E2 -12576.421} C_VEL
LIN {X 0,Y 368.929,Z 327.151,A -85,B 0,C 180,E1 -12579.946,E2 -12579.946} C_VEL
LIN {X 0,Y 368.968,Z 327.146,A -85,B 0,C 180,E1 -12583.398,E2 -12583.398} C_VEL
LIN {X 0,Y 369.05,Z 327.14,A -85,B 0,C 180,E1 -12586.79,E2 -12586.79} C_VEL
LIN {X 0,Y 369.06,Z 327.137,A -85,B 0,C 180,E1 -12590.131,E2 -12590.131} C_VEL
LIN {X 0,Y 369.181,Z 327.124,A -85,B 0,C 180,E1 -12592.342,E2 -12592.342} C_VEL
LIN {X 0,Y 369.138,Z 327.131,A -85,B 0,C 180,E1 -12594.537,E2 -12594.537} C_VEL
LIN {X 0,Y 369.312,Z 327.104,A -85,B 0,C 180,E1 -12597.818,E2 -12597.818} C_VEL
LIN {X 0,Y 369.45,Z 327.089,A -85,B 0,C 180,E1 -12600,E2 -12600} C_VEL
LIN {X 0,Y 369.311,Z 327.108,A -85,B 0,C 180,E1 -12602.181,E2 -12602.181} C_VEL
LIN {X 0,Y 369.2,Z 327.121,A -85,B 0,C 180,E1 -12606.558,E2 -12606.558} C_VEL
LIN {X 0,Y 369.131,Z 327.127,A -85,B 0,C 180,E1 -12608.761,E2 -12608.761} C_VEL
LIN {X 0,Y 369.005,Z 327.147,A -85,B 0,C 180,E1 -12612.093,E2 -12612.093} C_VEL
LIN {X 0,Y 368.993,Z 327.144,A -85,B 0,C 180,E1 -12615.465,E2 -12615.465} C_VEL
LIN {X 0,Y 368.974,Z 327.146,A -85,B 0,C 180,E1 -12618.893,E2 -12618.893} C_VEL
LIN {X 0,Y 368.924,Z 327.154,A -85,B 0,C 180,E1 -12622.395,E2 -12622.395} C_VEL
LIN {X 0,Y 368.992,Z 327.15,A -85,B 0,C 180,E1 -12625.981,E2 -12625.981} C_VEL
LIN {X 0,Y 368.96,Z 327.147,A -85,B 0,C 180,E1 -12628.814,E2 -12628.814} C_VEL
LIN {X 0,Y 368.903,Z 327.157,A -85,B 0,C 180,E1 -12632.237,E2 -12632.237} C_VEL
LIN {X 0,Y 368.922,Z 327.152,A -85,B 0,C 180,E1 -12635.002,E2 -12635.002} C_VEL
LIN {X 0,Y 368.907,Z 327.159,A -85,B 0,C 180,E1 -12638.642,E2 -12638.642} C_VEL
LIN {X 0,Y 368.975,Z 327.263,A -85,B 0,C 180,E1 -12640.522,E2 -12640.522} C_VEL
LIN {X 0,Y 370.573,Z 335.62,A -85,B 0,C 180,E1 -12643.891,E2 -12643.891} C_VEL
LIN {X 0,Y 372.465,Z 344.704,A -85,B 0,C 180,E1 -12647.382,E2 -12647.382} C_VEL
LIN {X 0,Y 373.551,Z 350.635,A -85,B 0,C 180,E1 -12649.566,E2 -12649.566} C_VEL
LIN {X 0,Y 373.291,Z 354.897,A -85,B 0,C 180,E1 -12651.031,E2 -12651.031} C_VEL
LIN {X 0,Y 371.925,Z 366.43,A -85,B 0,C 180,E1 -12654.872,E2 -12654.872} C_VEL
LIN {X 0,Y 370.757,Z 378.682,A -85,B 0,C 180,E1 -12658.865,E2 -12658.865} C_VEL
LIN {X 0,Y 369.736,Z 391.177,A -85,B 0,C 180,E1 -12662.859,E2 -12662.859} C_VEL
LIN {X 0,Y 369.061,Z 402.521,A -85,B 0,C 180,E1 -12666.429,E2 -12666.429} C_VEL
LIN {X 0,Y 368.922,Z 404.814,A -85,B 0,C 180,E1 -12667.088,E2 -12667.088} C_VEL
LIN {X 0,Y 369.184,Z 407.707,A -85,B 0,C 180,E1 -12667.249,E2 -12667.249} C_VEL
LIN {X 0,Y 371.009,Z 423.139,A -85,B 0,C 180,E1 -12667.914,E2 -12667.914} C_VEL
LIN {X 0,Y 372.689,Z 438.954,A -85,B 0,C 180,E1 -12668.832,E2 -12668.832} C_VEL
LIN {X 0,Y 373.647,Z 452.016,A -85,B 0,C 180,E1 -12669.782,E2 -12669.782} C_VEL
LIN {X 0,Y 372.697,Z 464.225,A -85,B 0,C 180,E1 -12670.816,E2 -12670.816} C_VEL
LIN {X 0,Y 371.573,Z 476.614,A -85,B 0,C 180,E1 -12672.101,E2 -12672.101} C_VEL
LIN {X 0,Y 370.408,Z 487.453,A -85,B 0,C 180,E1 -12673.466,E2 -12673.466} C_VEL
LIN {X 0,Y 369.448,Z 498.287,A -85,B 0,C 180,E1 -12675.12,E2 -12675.12} C_VEL
LIN {X 0,Y 368.798,Z 507.297,A -85,B 0,C 180,E1 -12676.782,E2 -12676.782} C_VEL
LIN {X 0,Y 368.359,Z 515.938,A -85,B 0,C 180,E1 -12678.724,E2 -12678.724} C_VEL
LIN {X 0,Y 368.155,Z 522.874,A -85,B 0,C 180,E1 -12680.663,E2 -12680.663} C_VEL
LIN {X 0,Y 368.201,Z 527.612,A -85,B 0,C 180,E1 -12682.323,E2 -12682.323} C_VEL
LIN {X 0,Y 368.358,Z 532.409,A -85,B 0,C 180,E1 -12684.527,E2 -12684.527} C_VEL
LIN {X 0,Y 368.417,Z 534.179,A -85,B 0,C 180,E1 -12685.625,E2 -12685.625} C_VEL
LIN {X 0,Y 368.448,Z 535.536,A -85,B 0,C 180,E1 -12686.721,E2 -12686.721} C_VEL
LIN {X 0,Y 368.663,Z 537.1,A -85,B 0,C 180,E1 -12688.909,E2 -12688.909} C_VEL
LIN {X 0,Y 368.848,Z 537.328,A -85,B 0,C 180,E1 -12690.001,E2 -12690.001} C_VEL
LIN {X 0,Y 368.722,Z 537.131,A -85,B 0,C 180,E1 -12691.093,E2 -12691.093} C_VEL
LIN {X 0,Y 368.449,Z 535.607,A -85,B 0,C 180,E1 -12693.281,E2 -12693.281} C_VEL
LIN {X 0,Y 368.476,Z 534.307,A -85,B 0,C 180,E1 -12694.376,E2 -12694.376} C_VEL
LIN {X 0,Y 368.214,Z 530.51,A -85,B 0,C 180,E1 -12696.577,E2 -12696.577} C_VEL
LIN {X 0,Y 368.069,Z 525.135,A -85,B 0,C 180,E1 -12698.787,E2 -12698.787} C_VEL
LIN {X 0,Y 368.21,Z 518.082,A -85,B 0,C 180,E1 -12701.004,E2 -12701.004} C_VEL
LIN {X 0,Y 368.601,Z 510.374,A -85,B 0,C 180,E1 -12702.947,E2 -12702.947} C_VEL
LIN {X 0,Y 369.447,Z 501.047,A -85,B 0,C 180,E1 -12704.882,E2 -12704.882} C_VEL
LIN {X 0,Y 370.658,Z 489.839,A -85,B 0,C 180,E1 -12706.808,E2 -12706.808} C_VEL
LIN {X 0,Y 372.258,Z 477.391,A -85,B 0,C 180,E1 -12708.579,E2 -12708.579} C_VEL
LIN {X 0,Y 374.072,Z 464.847,A -85,B 0,C 180,E1 -12710.051,E2 -12710.051} C_VEL
LIN {X 0,Y 375.392,Z 454.173,A -85,B 0,C 180,E1 -12711.125,E2 -12711.125} C_VEL
LIN {X 0,Y 375.729,Z 440.672,A -85,B 0,C 180,E1 -12712.37,E2 -12712.37} C_VEL
LIN {X 0,Y 375.762,Z 426.86,A -85,B 0,C 180,E1 -12713.474,E2 -12713.474} C_VEL
LIN {X 0,Y 374.269,Z 411.686,A -85,B 0,C 180,E1 -12714.634,E2 -12714.634} C_VEL
LIN {X 0,Y 371.775,Z 398.129,A -85,B 0,C 180,E1 -12715.667,E2 -12715.667} C_VEL
LIN {X 0,Y 369.821,Z 390.363,A -85,B 0,C 180,E1 -12716.279,E2 -12716.279} C_VEL
LIN {X 0,Y 369.134,Z 386.822,A -85,B 0,C 180,E1 -12716.583,E2 -12716.583} C_VEL
LIN {X 0,Y 369.287,Z 382.63,A -85,B 0,C 180,E1 -12717.793,E2 -12717.793} C_VEL
LIN {X 0,Y 369.887,Z 372.992,A -85,B 0,C 180,E1 -12720.865,E2 -12720.865} C_VEL
LIN {X 0,Y 370.759,Z 361.851,A -85,B 0,C 180,E1 -12724.659,E2 -12724.659} C_VEL
LIN {X 0,Y 372.389,Z 351.4,A -85,B 0,C 180,E1 -12728.522,E2 -12728.522} C_VEL
LIN {X 0,Y 372.995,Z 348.109,A -85,B 0,C 180,E1 -12729.84,E2 -12729.84} C_VEL
LIN {X 0,Y 372.399,Z 343.636,A -85,B 0,C 180,E1 -12731.947,E2 -12731.947} C_VEL
LIN {X 0,Y 371.487,Z 339.042,A -85,B 0,C 180,E1 -12734.427,E2 -12734.427} C_VEL
LIN {X 0,Y 370.374,Z 333.925,A -85,B 0,C 180,E1 -12737.736,E2 -12737.736} C_VEL
LIN {X 0,Y 369.844,Z 331.347,A -85,B 0,C 180,E1 -12739.753,E2 -12739.753} C_VEL
LIN {X 0,Y 369.043,Z 327.908,A -85,B 0,C 180,E1 -12743.116,E2 -12743.116} C_VEL
LIN {X 0,Y 368.905,Z 327.168,A -85,B 0,C 180,E1 -12744.127,E2 -12744.127} C_VEL
LIN {X 0,Y 368.901,Z 327.159,A -85,B 0,C 180,E1 -12747.763,E2 -12747.763} C_VEL
LIN {X 0,Y 368.966,Z 327.15,A -85,B 0,C 180,E1 -12751.563,E2 -12751.563} C_VEL
LIN {X 0,Y 368.966,Z 327.256,A -85,B 0,C 180,E1 -12752.797,E2 -12752.797} C_VEL
LIN {X 0,Y 369.222,Z 328.37,A -85,B 0,C 180,E1 -12753.088,E2 -12753.088} C_VEL
LIN {X 0,Y 373.172,Z 335.116,A -85,B 0,C 180,E1 -12754.169,E2 -12754.169} C_VEL
LIN {X 0,Y 378.733,Z 347.281,A -85,B 0,C 180,E1 -12755.906,E2 -12755.906} C_VEL
LIN {X 0,Y 382.146,Z 357.276,A -85,B 0,C 180,E1 -12757.281,E2 -12757.281} C_VEL
LIN {X 0,Y 382.382,Z 358.453,A -85,B 0,C 180,E1 -12757.434,E2 -12757.434} C_VEL
LIN {X 0,Y 380.66,Z 371.499,A -85,B 0,C 180,E1 -12758.757,E2 -12758.757} C_VEL
LIN {X 0,Y 379.246,Z 381.195,A -85,B 0,C 180,E1 -12759.951,E2 -12759.951} C_VEL
LIN {X 0,Y 377.523,Z 392.056,A -85,B 0,C 180,E1 -12761.55,E2 -12761.55} C_VEL
LIN {X 0,Y 375.875,Z 401.059,A -85,B 0,C 180,E1 -12763.153,E2 -12763.153} C_VEL
LIN {X 0,Y 374.32,Z 409.607,A -85,B 0,C 180,E1 -12765.039,E2 -12765.039} C_VEL
LIN {X 0,Y 372.954,Z 416.552,A -85,B 0,C 180,E1 -12766.931,E2 -12766.931} C_VEL
LIN {X 0,Y 371.758,Z 422.755,A -85,B 0,C 180,E1 -12769.103,E2 -12769.103} C_VEL
LIN {X 0,Y 370.735,Z 427.358,A -85,B 0,C 180,E1 -12771.277,E2 -12771.277} C_VEL
LIN {X 0,Y 369.892,Z 430.466,A -85,B 0,C 180,E1 -12773.454,E2 -12773.454} C_VEL
LIN {X 0,Y 369.436,Z 432.16,A -85,B 0,C 180,E1 -12775.636,E2 -12775.636} C_VEL
LIN {X 0,Y 369.158,Z 432.529,A -85,B 0,C 180,E1 -12777.818,E2 -12777.818} C_VEL
LIN {X 0,Y 368.988,Z 431.568,A -85,B 0,C 180,E1 -12780,E2 -12780} C_VEL
LIN {X 0,Y 368.928,Z 429.263,A -85,B 0,C 180,E1 -12782.184,E2 -12782.184} C_VEL
LIN {X 0,Y 368.956,Z 425.567,A -85,B 0,C 180,E1 -12784.37,E2 -12784.37} C_VEL
LIN {X 0,Y 369.488,Z 420.29,A -85,B 0,C 180,E1 -12786.554,E2 -12786.554} C_VEL
LIN {X 0,Y 370.013,Z 413.378,A -85,B 0,C 180,E1 -12788.74,E2 -12788.74} C_VEL
LIN {X 0,Y 370.642,Z 405.776,A -85,B 0,C 180,E1 -12790.654,E2 -12790.654} C_VEL
LIN {X 0,Y 371.338,Z 397.873,A -85,B 0,C 180,E1 -12792.294,E2 -12792.294} C_VEL
LIN {X 0,Y 372.167,Z 388.451,A -85,B 0,C 180,E1 -12793.932,E2 -12793.932} C_VEL
LIN {X 0,Y 373.058,Z 379.116,A -85,B 0,C 180,E1 -12795.293,E2 -12795.293} C_VEL
LIN {X 0,Y 374.056,Z 366.894,A -85,B 0,C 180,E1 -12796.79,E2 -12796.79} C_VEL
LIN {X 0,Y 374.935,Z 354.676,A -85,B 0,C 180,E1 -12798.017,E2 -12798.017} C_VEL
LIN {X 0,Y 375.348,Z 350.066,A -85,B 0,C 180,E1 -12798.42,E2 -12798.42} C_VEL
LIN {X 0,Y 374.258,Z 345.136,A -85,B 0,C 180,E1 -12798.884,E2 -12798.884} C_VEL
LIN {X 0,Y 370.145,Z 331.344,A -85,B 0,C 180,E1 -12800.075,E2 -12800.075} C_VEL
LIN {X 0,Y 369.11,Z 327.827,A -85,B 0,C 180,E1 -12800.375,E2 -12800.375} C_VEL
LIN {X 0,Y 368.989,Z 327.188,A -85,B 0,C 180,E1 -12800.581,E2 -12800.581} C_VEL
LIN {X 0,Y 368.95,Z 327.152,A -85,B 0,C 180,E1 -12803.887,E2 -12803.887} C_VEL
LIN {X 0,Y 368.973,Z 327.147,A -85,B 0,C 180,E1 -12807.203,E2 -12807.203} C_VEL
LIN {X 0,Y 368.924,Z 327.152,A -85,B 0,C 180,E1 -12809.69,E2 -12809.69} C_VEL
LIN {X 0,Y 368.902,Z 327.156,A -85,B 0,C 180,E1 -12813.043,E2 -12813.043} C_VEL
LIN {X 0,Y 368.922,Z 327.155,A -85,B 0,C 180,E1 -12816.197,E2 -12816.197} C_VEL
LIN {X 0,Y 368.907,Z 327.156,A -85,B 0,C 180,E1 -12818.953,E2 -12818.953} C_VEL
LIN {X 0,Y 368.886,Z 327.158,A -85,B 0,C 180,E1 -12822.009,E2 -12822.009} C_VEL
LIN {X 0,Y 368.887,Z 327.157,A -85,B 0,C 180,E1 -12825.176,E2 -12825.176} C_VEL
LIN {X 0,Y 368.915,Z 327.157,A -85,B 0,C 180,E1 -12828.181,E2 -12828.181} C_VEL
LIN {X 0,Y 368.916,Z 327.153,A -85,B 0,C 180,E1 -12831.359,E2 -12831.359} C_VEL
LIN {X 0,Y 368.942,Z 327.149,A -85,B 0,C 180,E1 -12835.146,E2 -12835.146} C_VEL
LIN {X 0,Y 368.935,Z 327.15,A -85,B 0,C 180,E1 -12839.046,E2 -12839.046} C_VEL
LIN {X 0,Y 368.969,Z 327.147,A -85,B 0,C 180,E1 -12842.796,E2 -12842.796} C_VEL
LIN {X 0,Y 368.94,Z 327.156,A -85,B 0,C 180,E1 -12846.116,E2 -12846.116} C_VEL
LIN {X 0,Y 368.943,Z 327.155,A -85,B 0,C 180,E1 -12849.947,E2 -12849.947} C_VEL
LIN {X 0,Y 368.982,Z 327.145,A -85,B 0,C 180,E1 -12853.398,E2 -12853.398} C_VEL
LIN {X 0,Y 369.063,Z 327.134,A -85,B 0,C 180,E1 -12856.79,E2 -12856.79} C_VEL
LIN {X 0,Y 369.073,Z 327.137,A -85,B 0,C 180,E1 -12860.131,E2 -12860.131} C_VEL
LIN {X 0,Y 369.193,Z 327.12,A -85,B 0,C 180,E1 -12862.341,E2 -12862.341} C_VEL
LIN {X 0,Y 369.148,Z 327.124,A -85,B 0,C 180,E1 -12864.537,E2 -12864.537} C_VEL
LIN {X 0,Y 369.321,Z 327.108,A -85,B 0,C 180,E1 -12867.818,E2 -12867.818} C_VEL
LIN {X 0,Y 369.461,Z 327.088,A -85,B 0,C 180,E1 -12869.999,E2 -12869.999} C_VEL
LIN {X 0,Y 369.321,Z 327.104,A -85,B 0,C 180,E1 -12872.18,E2 -12872.18} C_VEL
LIN {X 0,Y 369.213,Z 327.116,A -85,B 0,C 180,E1 -12876.557,E2 -12876.557} C_VEL
LIN {X 0,Y 369.141,Z 327.125,A -85,B 0,C 180,E1 -12878.76,E2 -12878.76} C_VEL
LIN {X 0,Y 369.009,Z 327.142,A -85,B 0,C 180,E1 -12882.092,E2 -12882.092} C_VEL
LIN {X 0,Y 369,Z 327.148,A -85,B 0,C 180,E1 -12885.464,E2 -12885.464} C_VEL
LIN {X 0,Y 368.96,Z 327.148,A -85,B 0,C 180,E1 -12888.893,E2 -12888.893} C_VEL
LIN {X 0,Y 368.937,Z 327.15,A -85,B 0,C 180,E1 -12892.394,E2 -12892.394} C_VEL
LIN {X 0,Y 369.001,Z 327.143,A -85,B 0,C 180,E1 -12895.979,E2 -12895.979} C_VEL
LIN {X 0,Y 368.914,Z 327.155,A -85,B 0,C 180,E1 -12899.689,E2 -12899.689} C_VEL
LIN {X 0,Y 368.896,Z 327.159,A -85,B 0,C 180,E1 -12903.042,E2 -12903.042} C_VEL
LIN {X 0,Y 368.915,Z 327.153,A -85,B 0,C 180,E1 -12906.195,E2 -12906.195} C_VEL
LIN {X 0,Y 368.879,Z 327.156,A -85,B 0,C 180,E1 -12909.768,E2 -12909.768} C_VEL
LIN {X 0,Y 368.234,Z 327.241,A -85,B 0,C 180,E1 -12910.679,E2 -12910.679} C_VEL
LIN {X 0,Y 365.396,Z 327.593,A -85,B 0,C 180,E1 -12912.162,E2 -12912.162} C_VEL
LIN {X 0,Y 362.97,Z 327.897,A -85,B 0,C 180,E1 -12913.361,E2 -12913.361} C_VEL
LIN {X 0,Y 361.913,Z 328.026,A -85,B 0,C 180,E1 -12914.288,E2 -12914.288} C_VEL
LIN {X 0,Y 361.819,Z 328.036,A -85,B 0,C 180,E1 -12914.603,E2 -12914.603} C_VEL
LIN {X 0,Y 361.833,Z 328.036,A -85,B 0,C 180,E1 -12917.567,E2 -12917.567} C_VEL
LIN {X 0,Y 361.868,Z 328.037,A -85,B 0,C 180,E1 -12920.972,E2 -12920.972} C_VEL
LIN {X 0,Y 361.87,Z 328.034,A -85,B 0,C 180,E1 -12924.654,E2 -12924.654} C_VEL
LIN {X 0,Y 361.855,Z 328.034,A -85,B 0,C 180,E1 -12928.372,E2 -12928.372} C_VEL
LIN {X 0,Y 361.917,Z 328.026,A -85,B 0,C 180,E1 -12932.221,E2 -12932.221} C_VEL
LIN {X 0,Y 361.922,Z 328.03,A -85,B 0,C 180,E1 -12934.709,E2 -12934.709} C_VEL
LIN {X 0,Y 361.887,Z 328.031,A -85,B 0,C 180,E1 -12938.346,E2 -12938.346} C_VEL
LIN {X 0,Y 361.96,Z 328.02,A -85,B 0,C 180,E1 -12942.061,E2 -12942.061} C_VEL
LIN {X 0,Y 361.99,Z 328.017,A -85,B 0,C 180,E1 -12946.101,E2 -12946.101} C_VEL
LIN {X 0,Y 362.024,Z 328.012,A -85,B 0,C 180,E1 -12949.937,E2 -12949.937} C_VEL
LIN {X 0,Y 362.139,Z 328,A -85,B 0,C 180,E1 -12952.192,E2 -12952.192} C_VEL
LIN {X 0,Y 362.111,Z 328.006,A -85,B 0,C 180,E1 -12954.431,E2 -12954.431} C_VEL
LIN {X 0,Y 362.276,Z 327.981,A -85,B 0,C 180,E1 -12957.776,E2 -12957.776} C_VEL
LIN {X 0,Y 362.42,Z 327.964,A -85,B 0,C 180,E1 -12960,E2 -12960} C_VEL
LIN {X 0,Y 362.275,Z 327.985,A -85,B 0,C 180,E1 -12962.223,E2 -12962.223} C_VEL
LIN {X 0,Y 362.164,Z 327.996,A -85,B 0,C 180,E1 -12966.686,E2 -12966.686} C_VEL
LIN {X 0,Y 362.067,Z 328.006,A -85,B 0,C 180,E1 -12968.933,E2 -12968.933} C_VEL
LIN {X 0,Y 361.959,Z 328.024,A -85,B 0,C 180,E1 -12972.332,E2 -12972.332} C_VEL
LIN {X 0,Y 361.956,Z 328.022,A -85,B 0,C 180,E1 -12974.62,E2 -12974.62} C_VEL
LIN {X 0,Y 361.951,Z 328.027,A -85,B 0,C 180,E1 -12978.099,E2 -12978.099} C_VEL
LIN {X 0,Y 361.884,Z 328.031,A -85,B 0,C 180,E1 -12981.653,E2 -12981.653} C_VEL
LIN {X 0,Y 361.92,Z 328.025,A -85,B 0,C 180,E1 -12985.29,E2 -12985.29} C_VEL
LIN {X 0,Y 361.915,Z 328.029,A -85,B 0,C 180,E1 -12987.778,E2 -12987.778} C_VEL
LIN {X 0,Y 361.852,Z 328.036,A -85,B 0,C 180,E1 -12991.628,E2 -12991.628} C_VEL
LIN {X 0,Y 361.868,Z 328.032,A -85,B 0,C 180,E1 -12995.346,E2 -12995.346} C_VEL
LIN {X 0,Y 361.86,Z 328.037,A -85,B 0,C 180,E1 -12999.027,E2 -12999.027} C_VEL
LIN {X 0,Y 361.96,Z 328.26,A -85,B 0,C 180,E1 -13000.228,E2 -13000.228} C_VEL
LIN {X 0,Y 363.752,Z 337.648,A -85,B 0,C 180,E1 -13004.071,E2 -13004.071} C_VEL
LIN {X 0,Y 365.704,Z 347.05,A -85,B 0,C 180,E1 -13007.732,E2 -13007.732} C_VEL
LIN {X 0,Y 366.488,Z 351.264,A -85,B 0,C 180,E1 -13009.309,E2 -13009.309} C_VEL
LIN {X 0,Y 366.38,Z 355.264,A -85,B 0,C 180,E1 -13010.729,E2 -13010.729} C_VEL
LIN {X 0,Y 364.916,Z 366.964,A -85,B 0,C 180,E1 -13014.707,E2 -13014.707} C_VEL
LIN {X 0,Y 363.768,Z 378.529,A -85,B 0,C 180,E1 -13018.559,E2 -13018.559} C_VEL
LIN {X 0,Y 362.772,Z 389.948,A -85,B 0,C 180,E1 -13022.294,E2 -13022.294} C_VEL
LIN {X 0,Y 362.059,Z 401.246,A -85,B 0,C 180,E1 -13025.945,E2 -13025.945} C_VEL
LIN {X 0,Y 361.916,Z 404.064,A -85,B 0,C 180,E1 -13026.77,E2 -13026.77} C_VEL
LIN {X 0,Y 362.221,Z 407.576,A -85,B 0,C 180,E1 -13026.946,E2 -13026.946} C_VEL
LIN {X 0,Y 364.061,Z 423.437,A -85,B 0,C 180,E1 -13027.663,E2 -13027.663} C_VEL
LIN {X 0,Y 365.637,Z 438.689,A -85,B 0,C 180,E1 -13028.581,E2 -13028.581} C_VEL
LIN {X 0,Y 366.569,Z 451.242,A -85,B 0,C 180,E1 -13029.52,E2 -13029.52} C_VEL
LIN {X 0,Y 366.304,Z 457.858,A -85,B 0,C 180,E1 -13030.073,E2 -13030.073} C_VEL
LIN {X 0,Y 365.032,Z 470.8,A -85,B 0,C 180,E1 -13031.333,E2 -13031.333} C_VEL
LIN {X 0,Y 363.879,Z 482.463,A -85,B 0,C 180,E1 -13032.726,E2 -13032.726} C_VEL
LIN {X 0,Y 362.838,Z 493.128,A -85,B 0,C 180,E1 -13034.267,E2 -13034.267} C_VEL
LIN {X 0,Y 362.025,Z 502.652,A -85,B 0,C 180,E1 -13035.924,E2 -13035.924} C_VEL
LIN {X 0,Y 361.482,Z 510.907,A -85,B 0,C 180,E1 -13037.652,E2 -13037.652} C_VEL
LIN {X 0,Y 361.214,Z 517.633,A -85,B 0,C 180,E1 -13039.349,E2 -13039.349} C_VEL
LIN {X 0,Y 361.103,Z 523.177,A -85,B 0,C 180,E1 -13041.044,E2 -13041.044} C_VEL
LIN {X 0,Y 361.215,Z 528.004,A -85,B 0,C 180,E1 -13042.878,E2 -13042.878} C_VEL
LIN {X 0,Y 361.32,Z 531.142,A -85,B 0,C 180,E1 -13044.42,E2 -13044.42} C_VEL
LIN {X 0,Y 361.387,Z 532.943,A -85,B 0,C 180,E1 -13045.54,E2 -13045.54} C_VEL
LIN {X 0,Y 361.426,Z 534.341,A -85,B 0,C 180,E1 -13046.657,E2 -13046.657} C_VEL
LIN {X 0,Y 361.643,Z 535.987,A -85,B 0,C 180,E1 -13048.887,E2 -13048.887} C_VEL
LIN {X 0,Y 361.838,Z 536.24,A -85,B 0,C 180,E1 -13050.001,E2 -13050.001} C_VEL
LIN {X 0,Y 361.694,Z 536.062,A -85,B 0,C 180,E1 -13051.114,E2 -13051.114} C_VEL
LIN {X 0,Y 361.409,Z 534.583,A -85,B 0,C 180,E1 -13053.345,E2 -13053.345} C_VEL
LIN {X 0,Y 361.413,Z 533.297,A -85,B 0,C 180,E1 -13054.462,E2 -13054.462} C_VEL
LIN {X 0,Y 361.106,Z 529.543,A -85,B 0,C 180,E1 -13056.707,E2 -13056.707} C_VEL
LIN {X 0,Y 360.996,Z 524.22,A -85,B 0,C 180,E1 -13058.961,E2 -13058.961} C_VEL
LIN {X 0,Y 361.177,Z 517.245,A -85,B 0,C 180,E1 -13061.221,E2 -13061.221} C_VEL
LIN {X 0,Y 361.557,Z 509.633,A -85,B 0,C 180,E1 -13063.204,E2 -13063.204} C_VEL
LIN {X 0,Y 362.497,Z 500.467,A -85,B 0,C 180,E1 -13065.174,E2 -13065.174} C_VEL
LIN {X 0,Y 363.811,Z 489.417,A -85,B 0,C 180,E1 -13067.134,E2 -13067.134} C_VEL
LIN {X 0,Y 365.484,Z 477.182,A -85,B 0,C 180,E1 -13068.936,E2 -13068.936} C_VEL
LIN {X 0,Y 367.51,Z 464.351,A -85,B 0,C 180,E1 -13070.5,E2 -13070.5} C_VEL
LIN {X 0,Y 368.72,Z 454.582,A -85,B 0,C 180,E1 -13071.526,E2 -13071.526} C_VEL
LIN {X 0,Y 369.326,Z 439.864,A -85,B 0,C 180,E1 -13072.94,E2 -13072.94} C_VEL
LIN {X 0,Y 369.345,Z 425.498,A -85,B 0,C 180,E1 -13074.149,E2 -13074.149} C_VEL
LIN {X 0,Y 367.932,Z 411.391,A -85,B 0,C 180,E1 -13075.304,E2 -13075.304} C_VEL
LIN {X 0,Y 365.602,Z 398.772,A -85,B 0,C 180,E1 -13076.345,E2 -13076.345} C_VEL
LIN {X 0,Y 363.261,Z 389.022,A -85,B 0,C 180,E1 -13077.18,E2 -13077.18} C_VEL
LIN {X 0,Y 362.251,Z 384.609,A -85,B 0,C 180,E1 -13077.599,E2 -13077.599} C_VEL
LIN {X 0,Y 362.357,Z 381.912,A -85,B 0,C 180,E1 -13078.372,E2 -13078.372} C_VEL
LIN {X 0,Y 363.03,Z 372.17,A -85,B 0,C 180,E1 -13081.591,E2 -13081.591} C_VEL
LIN {X 0,Y 364.042,Z 361.417,A -85,B 0,C 180,E1 -13085.393,E2 -13085.393} C_VEL
LIN {X 0,Y 365.888,Z 351.205,A -85,B 0,C 180,E1 -13089.337,E2 -13089.337} C_VEL
LIN {X 0,Y 366.089,Z 349.156,A -85,B 0,C 180,E1 -13090.215,E2 -13090.215} C_VEL
LIN {X 0,Y 365.183,Z 343.606,A -85,B 0,C 180,E1 -13093.003,E2 -13093.003} C_VEL
LIN {X 0,Y 364.154,Z 338.582,A -85,B 0,C 180,E1 -13095.99,E2 -13095.99} C_VEL
LIN {X 0,Y 363.254,Z 334.43,A -85,B 0,C 180,E1 -13098.987,E2 -13098.987} C_VEL
LIN {X 0,Y 362.621,Z 331.425,A -85,B 0,C 180,E1 -13101.67,E2 -13101.67} C_VEL
LIN {X 0,Y 362.033,Z 328.855,A -85,B 0,C 180,E1 -13104.621,E2 -13104.621} C_VEL
LIN {X 0,Y 361.876,Z 328.076,A -85,B 0,C 180,E1 -13105.722,E2 -13105.722} C_VEL
LIN {X 0,Y 361.876,Z 328.035,A -85,B 0,C 180,E1 -13109.672,E2 -13109.672} C_VEL
LIN {X 0,Y 361.941,Z 328.151,A -85,B 0,C 180,E1 -13111.672,E2 -13111.672} C_VEL
LIN {X 0,Y 362.246,Z 329.471,A -85,B 0,C 180,E1 -13112.012,E2 -13112.012} C_VEL
LIN {X 0,Y 363.203,Z 331.3,A -85,B 0,C 180,E1 -13112.329,E2 -13112.329} C_VEL
LIN {X 0,Y 364.833,Z 333.668,A -85,B 0,C 180,E1 -13112.777,E2 -13112.777} C_VEL
LIN {X 0,Y 369.902,Z 343.095,A -85,B 0,C 180,E1 -13114.33,E2 -13114.33} C_VEL
LIN {X 0,Y 373.823,Z 352.573,A -85,B 0,C 180,E1 -13115.76,E2 -13115.76} C_VEL
LIN {X 0,Y 376.302,Z 360.476,A -85,B 0,C 180,E1 -13116.908,E2 -13116.908} C_VEL
LIN {X 0,Y 374.626,Z 373.175,A -85,B 0,C 180,E1 -13118.253,E2 -13118.253} C_VEL
LIN {X 0,Y 372.95,Z 383.735,A -85,B 0,C 180,E1 -13119.597,E2 -13119.597} C_VEL
LIN {X 0,Y 371.072,Z 394.547,A -85,B 0,C 180,E1 -13121.262,E2 -13121.262} C_VEL
LIN {X 0,Y 369.049,Z 404.39,A -85,B 0,C 180,E1 -13123.117,E2 -13123.117} C_VEL
LIN {X 0,Y 367.489,Z 412.527,A -85,B 0,C 180,E1 -13125.038,E2 -13125.038} C_VEL
LIN {X 0,Y 366.243,Z 418.251,A -85,B 0,C 180,E1 -13126.687,E2 -13126.687} C_VEL
LIN {X 0,Y 364.977,Z 424.322,A -85,B 0,C 180,E1 -13128.898,E2 -13128.898} C_VEL
LIN {X 0,Y 363.86,Z 428.782,A -85,B 0,C 180,E1 -13131.111,E2 -13131.111} C_VEL
LIN {X 0,Y 362.961,Z 431.788,A -85,B 0,C 180,E1 -13133.329,E2 -13133.329} C_VEL
LIN {X 0,Y 362.478,Z 433.384,A -85,B 0,C 180,E1 -13135.552,E2 -13135.552} C_VEL
LIN {X 0,Y 362.153,Z 433.663,A -85,B 0,C 180,E1 -13137.776,E2 -13137.776} C_VEL
LIN {X 0,Y 361.971,Z 432.606,A -85,B 0,C 180,E1 -13140,E2 -13140} C_VEL
LIN {X 0,Y 361.903,Z 430.21,A -85,B 0,C 180,E1 -13142.226,E2 -13142.226} C_VEL
LIN {X 0,Y 361.854,Z 427.469,A -85,B 0,C 180,E1 -13143.898,E2 -13143.898} C_VEL
LIN {X 0,Y 362.205,Z 423.893,A -85,B 0,C 180,E1 -13145.568,E2 -13145.568} C_VEL
LIN {X 0,Y 362.745,Z 417.719,A -85,B 0,C 180,E1 -13147.795,E2 -13147.795} C_VEL
LIN {X 0,Y 363.28,Z 410.87,A -85,B 0,C 180,E1 -13149.746,E2 -13149.746} C_VEL
LIN {X 0,Y 364.051,Z 402.441,A -85,B 0,C 180,E1 -13151.695,E2 -13151.695} C_VEL
LIN {X 0,Y 364.813,Z 393.692,A -85,B 0,C 180,E1 -13153.367,E2 -13153.367} C_VEL
LIN {X 0,Y 365.758,Z 383.19,A -85,B 0,C 180,E1 -13155.035,E2 -13155.035} C_VEL
LIN {X 0,Y 366.795,Z 372.3,A -85,B 0,C 180,E1 -13156.471,E2 -13156.471} C_VEL
LIN {X 0,Y 367.748,Z 360.167,A -85,B 0,C 180,E1 -13157.805,E2 -13157.805} C_VEL
LIN {X 0,Y 368.448,Z 351.295,A -85,B 0,C 180,E1 -13158.633,E2 -13158.633} C_VEL
LIN {X 0,Y 365.648,Z 340.668,A -85,B 0,C 180,E1 -13159.64,E2 -13159.64} C_VEL
LIN {X 0,Y 362.046,Z 328.719,A -85,B 0,C 180,E1 -13160.666,E2 -13160.666} C_VEL
LIN {X 0,Y 361.922,Z 328.065,A -85,B 0,C 180,E1 -13160.887,E2 -13160.887} C_VEL
LIN {X 0,Y 361.901,Z 328.031,A -85,B 0,C 180,E1 -13164.114,E2 -13164.114} C_VEL
LIN {X 0,Y 361.948,Z 328.027,A -85,B 0,C 180,E1 -13166.722,E2 -13166.722} C_VEL
LIN {X 0,Y 361.88,Z 328.032,A -85,B 0,C 180,E1 -13170.328,E2 -13170.328} C_VEL
LIN {X 0,Y 361.859,Z 328.035,A -85,B 0,C 180,E1 -13174.28,E2 -13174.28} C_VEL
LIN {X 0,Y 361.868,Z 328.031,A -85,B 0,C 180,E1 -13177.223,E2 -13177.223} C_VEL
LIN {X 0,Y 361.841,Z 328.038,A -85,B 0,C 180,E1 -13180.755,E2 -13180.755} C_VEL
LIN {X 0,Y 361.824,Z 328.042,A -85,B 0,C 180,E1 -13184.368,E2 -13184.368} C_VEL
LIN {X 0,Y 361.862,Z 328.032,A -85,B 0,C 180,E1 -13187.564,E2 -13187.564} C_VEL
LIN {X 0,Y 361.878,Z 328.03,A -85,B 0,C 180,E1 -13190.973,E2 -13190.973} C_VEL
LIN {X 0,Y 361.88,Z 328.032,A -85,B 0,C 180,E1 -13194.655,E2 -13194.655} C_VEL
LIN {X 0,Y 361.844,Z 328.038,A -85,B 0,C 180,E1 -13198.37,E2 -13198.37} C_VEL
LIN {X 0,Y 361.914,Z 328.031,A -85,B 0,C 180,E1 -13202.221,E2 -13202.221} C_VEL
LIN {X 0,Y 361.932,Z 328.024,A -85,B 0,C 180,E1 -13204.709,E2 -13204.709} C_VEL
LIN {X 0,Y 361.867,Z 328.034,A -85,B 0,C 180,E1 -13208.345,E2 -13208.345} C_VEL
LIN {X 0,Y 361.973,Z 328.024,A -85,B 0,C 180,E1 -13212.061,E2 -13212.061} C_VEL
LIN {X 0,Y 362.003,Z 328.019,A -85,B 0,C 180,E1 -13216.1,E2 -13216.1} C_VEL
LIN {X 0,Y 362.037,Z 328.016,A -85,B 0,C 180,E1 -13219.937,E2 -13219.937} C_VEL
LIN {X 0,Y 362.156,Z 327.998,A -85,B 0,C 180,E1 -13222.192,E2 -13222.192} C_VEL
LIN {X 0,Y 362.122,Z 328,A -85,B 0,C 180,E1 -13224.43,E2 -13224.43} C_VEL
LIN {X 0,Y 362.285,Z 327.985,A -85,B 0,C 180,E1 -13227.775,E2 -13227.775} C_VEL
LIN {X 0,Y 362.431,Z 327.964,A -85,B 0,C 180,E1 -13229.999,E2 -13229.999} C_VEL
LIN {X 0,Y 362.285,Z 327.98,A -85,B 0,C 180,E1 -13232.223,E2 -13232.223} C_VEL
LIN {X 0,Y 362.176,Z 327.992,A -85,B 0,C 180,E1 -13236.685,E2 -13236.685} C_VEL
LIN {X 0,Y 362.078,Z 328.005,A -85,B 0,C 180,E1 -13238.932,E2 -13238.932} C_VEL
LIN {X 0,Y 361.963,Z 328.019,A -85,B 0,C 180,E1 -13242.331,E2 -13242.331} C_VEL
LIN {X 0,Y 361.964,Z 328.019,A -85,B 0,C 180,E1 -13244.619,E2 -13244.619} C_VEL
LIN {X 0,Y 361.958,Z 328.02,A -85,B 0,C 180,E1 -13248.098,E2 -13248.098} C_VEL
LIN {X 0,Y 361.895,Z 328.031,A -85,B 0,C 180,E1 -13251.651,E2 -13251.651} C_VEL
LIN {X 0,Y 361.929,Z 328.029,A -85,B 0,C 180,E1 -13255.289,E2 -13255.289} C_VEL
LIN {X 0,Y 361.908,Z 328.028,A -85,B 0,C 180,E1 -13257.778,E2 -13257.778} C_VEL
LIN {X 0,Y 361.837,Z 328.037,A -85,B 0,C 180,E1 -13261.628,E2 -13261.628} C_VEL
LIN {X 0,Y 361.873,Z 328.035,A -85,B 0,C 180,E1 -13265.343,E2 -13265.343} C_VEL
LIN {X 0,Y 361.868,Z 328.036,A -85,B 0,C 180,E1 -13269.025,E2 -13269.025} C_VEL
LIN {X 0,Y 361.834,Z 328.038,A -85,B 0,C 180,E1 -13272.827,E2 -13272.827} C_VEL
LIN {X 0,Y 361.819,Z 328.036,A -85,B 0,C 180,E1 -13274.603,E2 -13274.603} C_VEL
LIN {X 0,Y 361.133,Z 328.124,A -85,B 0,C 180,E1 -13275.532,E2 -13275.532} C_VEL
LIN {X 0,Y 358.286,Z 328.483,A -85,B 0,C 180,E1 -13277.044,E2 -13277.044} C_VEL
LIN {X 0,Y 355.887,Z 328.783,A -85,B 0,C 180,E1 -13278.267,E2 -13278.267} C_VEL
LIN {X 0,Y 354.858,Z 328.908,A -85,B 0,C 180,E1 -13279.213,E2 -13279.213} C_VEL
LIN {X 0,Y 354.774,Z 328.916,A -85,B 0,C 180,E1 -13279.533,E2 -13279.533} C_VEL
LIN {X 0,Y 354.804,Z 328.912,A -85,B 0,C 180,E1 -13282.401,E2 -13282.401} C_VEL
LIN {X 0,Y 354.808,Z 328.916,A -85,B 0,C 180,E1 -13284.94,E2 -13284.94} C_VEL
LIN {X 0,Y 354.81,Z 328.912,A -85,B 0,C 180,E1 -13288.398,E2 -13288.398} C_VEL
LIN {X 0,Y 354.849,Z 328.905,A -85,B 0,C 180,E1 -13291.618,E2 -13291.618} C_VEL
LIN {X 0,Y 354.893,Z 328.9,A -85,B 0,C 180,E1 -13294.172,E2 -13294.172} C_VEL
LIN {X 0,Y 354.829,Z 328.908,A -85,B 0,C 180,E1 -13297.893,E2 -13297.893} C_VEL
LIN {X 0,Y 354.915,Z 328.897,A -85,B 0,C 180,E1 -13301.891,E2 -13301.891} C_VEL
LIN {X 0,Y 354.935,Z 328.895,A -85,B 0,C 180,E1 -13305.98,E2 -13305.98} C_VEL
LIN {X 0,Y 354.971,Z 328.89,A -85,B 0,C 180,E1 -13309.735,E2 -13309.735} C_VEL
LIN {X 0,Y 355.121,Z 328.873,A -85,B 0,C 180,E1 -13312.037,E2 -13312.037} C_VEL
LIN {X 0,Y 355.085,Z 328.88,A -85,B 0,C 180,E1 -13314.32,E2 -13314.32} C_VEL
LIN {X 0,Y 355.239,Z 328.857,A -85,B 0,C 180,E1 -13317.732,E2 -13317.732} C_VEL
LIN {X 0,Y 355.39,Z 328.84,A -85,B 0,C 180,E1 -13320,E2 -13320} C_VEL
LIN {X 0,Y 355.238,Z 328.862,A -85,B 0,C 180,E1 -13322.267,E2 -13322.267} C_VEL
LIN {X 0,Y 355.13,Z 328.871,A -85,B 0,C 180,E1 -13326.819,E2 -13326.819} C_VEL
LIN {X 0,Y 355.009,Z 328.885,A -85,B 0,C 180,E1 -13329.112,E2 -13329.112} C_VEL
LIN {X 0,Y 354.918,Z 328.899,A -85,B 0,C 180,E1 -13332.581,E2 -13332.581} C_VEL
LIN {X 0,Y 354.884,Z 328.907,A -85,B 0,C 180,E1 -13336.096,E2 -13336.096} C_VEL
LIN {X 0,Y 354.898,Z 328.901,A -85,B 0,C 180,E1 -13338.472,E2 -13338.472} C_VEL
LIN {X 0,Y 354.827,Z 328.914,A -85,B 0,C 180,E1 -13342.106,E2 -13342.106} C_VEL
LIN {X 0,Y 354.892,Z 328.904,A -85,B 0,C 180,E1 -13345.828,E2 -13345.828} C_VEL
LIN {X 0,Y 354.847,Z 328.909,A -85,B 0,C 180,E1 -13349.679,E2 -13349.679} C_VEL
LIN {X 0,Y 354.823,Z 328.912,A -85,B 0,C 180,E1 -13353.683,E2 -13353.683} C_VEL
LIN {X 0,Y 354.795,Z 328.917,A -85,B 0,C 180,E1 -13356.46,E2 -13356.46} C_VEL
LIN {X 0,Y 354.878,Z 329.046,A -85,B 0,C 180,E1 -13359.831,E2 -13359.831} C_VEL
LIN {X 0,Y 356.618,Z 338.061,A -85,B 0,C 180,E1 -13363.611,E2 -13363.611} C_VEL
LIN {X 0,Y 358.506,Z 347.349,A -85,B 0,C 180,E1 -13367.318,E2 -13367.318} C_VEL
LIN {X 0,Y 359.415,Z 351.868,A -85,B 0,C 180,E1 -13369.048,E2 -13369.048} C_VEL
LIN {X 0,Y 359.562,Z 353.997,A -85,B 0,C 180,E1 -13369.835,E2 -13369.835} C_VEL
LIN {X 0,Y 358.595,Z 361.827,A -85,B 0,C 180,E1 -13372.588,E2 -13372.588} C_VEL
LIN {X 0,Y 357.503,Z 370.737,A -85,B 0,C 180,E1 -13375.655,E2 -13375.655} C_VEL
LIN {X 0,Y 356.523,Z 381.093,A -85,B 0,C 180,E1 -13379.169,E2 -13379.169} C_VEL
LIN {X 0,Y 355.546,Z 392.472,A -85,B 0,C 180,E1 -13382.96,E2 -13382.96} C_VEL
LIN {X 0,Y 354.903,Z 403.03,A -85,B 0,C 180,E1 -13386.399,E2 -13386.399} C_VEL
LIN {X 0,Y 355.068,Z 405.5,A -85,B 0,C 180,E1 -13386.565,E2 -13386.565} C_VEL
LIN {X 0,Y 356.777,Z 420.922,A -85,B 0,C 180,E1 -13387.257,E2 -13387.257} C_VEL
LIN {X 0,Y 358.396,Z 436.578,A -85,B 0,C 180,E1 -13388.202,E2 -13388.202} C_VEL
LIN {X 0,Y 359.357,Z 448.417,A -85,B 0,C 180,E1 -13389.09,E2 -13389.09} C_VEL
LIN {X 0,Y 359.54,Z 455.706,A -85,B 0,C 180,E1 -13389.711,E2 -13389.711} C_VEL
LIN {X 0,Y 358.254,Z 468.655,A -85,B 0,C 180,E1 -13390.967,E2 -13390.967} C_VEL
LIN {X 0,Y 357.006,Z 480.495,A -85,B 0,C 180,E1 -13392.383,E2 -13392.383} C_VEL
LIN {X 0,Y 355.909,Z 491.304,A -85,B 0,C 180,E1 -13393.953,E2 -13393.953} C_VEL
LIN {X 0,Y 355.005,Z 501.376,A -85,B 0,C 180,E1 -13395.724,E2 -13395.724} C_VEL
LIN {X 0,Y 354.405,Z 510.554,A -85,B 0,C 180,E1 -13397.693,E2 -13397.693} C_VEL
LIN {X 0,Y 354.094,Z 518.161,A -85,B 0,C 180,E1 -13399.711,E2 -13399.711} C_VEL
LIN {X 0,Y 354.08,Z 523.398,A -85,B 0,C 180,E1 -13401.44,E2 -13401.44} C_VEL
LIN {X 0,Y 354.175,Z 527.596,A -85,B 0,C 180,E1 -13403.163,E2 -13403.163} C_VEL
LIN {X 0,Y 354.281,Z 529.855,A -85,B 0,C 180,E1 -13404.309,E2 -13404.309} C_VEL
LIN {X 0,Y 354.357,Z 531.691,A -85,B 0,C 180,E1 -13405.451,E2 -13405.451} C_VEL
LIN {X 0,Y 354.488,Z 534.166,A -85,B 0,C 180,E1 -13407.729,E2 -13407.729} C_VEL
LIN {X 0,Y 354.826,Z 535.134,A -85,B 0,C 180,E1 -13410.001,E2 -13410.001} C_VEL
LIN {X 0,Y 354.665,Z 534.989,A -85,B 0,C 180,E1 -13411.136,E2 -13411.136} C_VEL
LIN {X 0,Y 354.366,Z 533.558,A -85,B 0,C 180,E1 -13413.412,E2 -13413.412} C_VEL
LIN {X 0,Y 354.335,Z 532.295,A -85,B 0,C 180,E1 -13414.551,E2 -13414.551} C_VEL
LIN {X 0,Y 354.049,Z 528.592,A -85,B 0,C 180,E1 -13416.841,E2 -13416.841} C_VEL
LIN {X 0,Y 353.903,Z 523.324,A -85,B 0,C 180,E1 -13419.142,E2 -13419.142} C_VEL
LIN {X 0,Y 354.143,Z 516.431,A -85,B 0,C 180,E1 -13421.447,E2 -13421.447} C_VEL
LIN {X 0,Y 354.519,Z 508.92,A -85,B 0,C 180,E1 -13423.471,E2 -13423.471} C_VEL
LIN {X 0,Y 355.562,Z 499.901,A -85,B 0,C 180,E1 -13425.477,E2 -13425.477} C_VEL
LIN {X 0,Y 356.965,Z 489.079,A -85,B 0,C 180,E1 -13427.473,E2 -13427.473} C_VEL
LIN {X 0,Y 358.744,Z 477.075,A -85,B 0,C 180,E1 -13429.306,E2 -13429.306} C_VEL
LIN {X 0,Y 360.912,Z 464.299,A -85,B 0,C 180,E1 -13430.922,E2 -13430.922} C_VEL
LIN {X 0,Y 362.118,Z 455.135,A -85,B 0,C 180,E1 -13431.939,E2 -13431.939} C_VEL
LIN {X 0,Y 362.89,Z 440.734,A -85,B 0,C 180,E1 -13433.393,E2 -13433.393} C_VEL
LIN {X 0,Y 363.084,Z 426.931,A -85,B 0,C 180,E1 -13434.627,E2 -13434.627} C_VEL
LIN {X 0,Y 361.656,Z 411.212,A -85,B 0,C 180,E1 -13436.005,E2 -13436.005} C_VEL
LIN {X 0,Y 359.114,Z 397.243,A -85,B 0,C 180,E1 -13437.258,E2 -13437.258} C_VEL
LIN {X 0,Y 356.523,Z 386.995,A -85,B 0,C 180,E1 -13438.237,E2 -13438.237} C_VEL
LIN {X 0,Y 355.442,Z 382.242,A -85,B 0,C 180,E1 -13438.733,E2 -13438.733} C_VEL
LIN {X 0,Y 355.616,Z 379.343,A -85,B 0,C 180,E1 -13439.61,E2 -13439.61} C_VEL
LIN {X 0,Y 356.495,Z 368.18,A -85,B 0,C 180,E1 -13443.505,E2 -13443.505} C_VEL
